LIN {X 0,Y 566.944,Z 607.654,A -85,B 0,C 180,E1 -2597.403,E2 -2597.403} C_VEL
LIN {X 0,Y 566.869,Z 619.609,A -85,B 0,C 180,E1 -2597.674,E2 -2597.674} C_VEL
LIN {X 0,Y 566.746,Z 633.413,A -85,B 0,C 180,E1 -2598.148,E2 -2598.148} C_VEL
LIN {X 0,Y 566.629,Z 645.045,A -85,B 0,C 180,E1 -2598.706,E2 -2598.706} C_VEL
LIN {X 0,Y 566.485,Z 655.838,A -85,B 0,C 180,E1 -2599.366,E2 -2599.366} C_VEL
LIN {X 0,Y 566.315,Z 665.418,A -85,B 0,C 180,E1 -2600.085,E2 -2600.085} C_VEL
LIN {X 0,Y 566.229,Z 674.312,A -85,B 0,C 180,E1 -2600.895,E2 -2600.895} C_VEL
LIN {X 0,Y 566.113,Z 683.962,A -85,B 0,C 180,E1 -2601.972,E2 -2601.972} C_VEL
LIN {X 0,Y 566.009,Z 691.72,A -85,B 0,C 180,E1 -2603.065,E2 -2603.065} C_VEL
LIN {X 0,Y 565.989,Z 696.846,A -85,B 0,C 180,E1 -2603.941,E2 -2603.941} C_VEL
LIN {X 0,Y 565.877,Z 701.915,A -85,B 0,C 180,E1 -2605.013,E2 -2605.013} C_VEL
LIN {X 0,Y 565.927,Z 705.855,A -85,B 0,C 180,E1 -2606.084,E2 -2606.084} C_VEL
LIN {X 0,Y 565.878,Z 708.77,A -85,B 0,C 180,E1 -2607.152,E2 -2607.152} C_VEL
LIN {X 0,Y 565.84,Z 710.209,A -85,B 0,C 180,E1 -2607.865,E2 -2607.865} C_VEL
LIN {X 0,Y 565.841,Z 711.767,A -85,B 0,C 180,E1 -2609.288,E2 -2609.288} C_VEL
LIN {X 0,Y 565.839,Z 712,A -85,B 0,C 180,E1 -2610,E2 -2610} C_VEL
LIN {X 0,Y 565.846,Z 711.177,A -85,B 0,C 180,E1 -2611.423,E2 -2611.423} C_VEL
LIN {X 0,Y 565.84,Z 710.209,A -85,B 0,C 180,E1 -2612.135,E2 -2612.135} C_VEL
LIN {X 0,Y 565.927,Z 706.934,A -85,B 0,C 180,E1 -2613.56,E2 -2613.56} C_VEL
LIN {X 0,Y 565.933,Z 703.334,A -85,B 0,C 180,E1 -2614.63,E2 -2614.63} C_VEL
LIN {X 0,Y 565.998,Z 698.641,A -85,B 0,C 180,E1 -2615.701,E2 -2615.701} C_VEL
LIN {X 0,Y 565.998,Z 692.926,A -85,B 0,C 180,E1 -2616.739,E2 -2616.739} C_VEL
LIN {X 0,Y 566.081,Z 686.651,A -85,B 0,C 180,E1 -2617.67,E2 -2617.67} C_VEL
LIN {X 0,Y 566.174,Z 679.383,A -85,B 0,C 180,E1 -2618.566,E2 -2618.566} C_VEL
LIN {X 0,Y 566.28,Z 670.607,A -85,B 0,C 180,E1 -2619.465,E2 -2619.465} C_VEL
LIN {X 0,Y 566.439,Z 659.729,A -85,B 0,C 180,E1 -2620.364,E2 -2620.364} C_VEL
LIN {X 0,Y 566.591,Z 649.221,A -85,B 0,C 180,E1 -2621.056,E2 -2621.056} C_VEL
LIN {X 0,Y 566.69,Z 638.78,A -85,B 0,C 180,E1 -2621.608,E2 -2621.608} C_VEL
LIN {X 0,Y 566.763,Z 628.631,A -85,B 0,C 180,E1 -2622.033,E2 -2622.033} C_VEL
LIN {X 0,Y 566.923,Z 617.028,A -85,B 0,C 180,E1 -2622.393,E2 -2622.393} C_VEL
LIN {X 0,Y 566.934,Z 605.012,A -85,B 0,C 180,E1 -2622.643,E2 -2622.643} C_VEL
LIN {X 0,Y 567.085,Z 506.315,A -85,B 0,C 180,E1 -2623.906,E2 -2623.906} C_VEL
LIN {X 0,Y 566.329,Z 501.567,A -85,B 0,C 180,E1 -2624.004,E2 -2624.004} C_VEL
LIN {X 0,Y 566.263,Z 499.133,A -85,B 0,C 180,E1 -2624.372,E2 -2624.372} C_VEL
LIN {X 0,Y 566.412,Z 482.577,A -85,B 0,C 180,E1 -2627.325,E2 -2627.325} C_VEL
LIN {X 0,Y 566.641,Z 467.055,A -85,B 0,C 180,E1 -2630.132,E2 -2630.132} C_VEL
LIN {X 0,Y 566.814,Z 451.485,A -85,B 0,C 180,E1 -2632.99,E2 -2632.99} C_VEL
LIN {X 0,Y 566.824,Z 444.171,A -85,B 0,C 180,E1 -2634.347,E2 -2634.347} C_VEL
LIN {X 0,Y 566.177,Z 440.526,A -85,B 0,C 180,E1 -2635.096,E2 -2635.096} C_VEL
LIN {X 0,Y 566.151,Z 440.46,A -85,B 0,C 180,E1 -2637.342,E2 -2637.342} C_VEL
LIN {X 0,Y 566.156,Z 440.462,A -85,B 0,C 180,E1 -2639.771,E2 -2639.771} C_VEL
LIN {X 0,Y 566.178,Z 440.458,A -85,B 0,C 180,E1 -2642.425,E2 -2642.425} C_VEL
LIN {X 0,Y 566.159,Z 440.456,A -85,B 0,C 180,E1 -2644.985,E2 -2644.985} C_VEL
LIN {X 0,Y 566.18,Z 440.454,A -85,B 0,C 180,E1 -2647.462,E2 -2647.462} C_VEL
LIN {X 0,Y 566.159,Z 440.461,A -85,B 0,C 180,E1 -2650.203,E2 -2650.203} C_VEL
LIN {X 0,Y 566.145,Z 440.458,A -85,B 0,C 180,E1 -2653.059,E2 -2653.059} C_VEL
LIN {X 0,Y 566.144,Z 440.466,A -85,B 0,C 180,E1 -2656.054,E2 -2656.054} C_VEL
LIN {X 0,Y 566.133,Z 440.459,A -85,B 0,C 180,E1 -2658.856,E2 -2658.856} C_VEL
LIN {X 0,Y 566.159,Z 440.458,A -85,B 0,C 180,E1 -2661.634,E2 -2661.634} C_VEL
LIN {X 0,Y 566.134,Z 440.464,A -85,B 0,C 180,E1 -2664.305,E2 -2664.305} C_VEL
LIN {X 0,Y 566.16,Z 440.455,A -85,B 0,C 180,E1 -2666.893,E2 -2666.893} C_VEL
LIN {X 0,Y 566.162,Z 440.457,A -85,B 0,C 180,E1 -2669.405,E2 -2669.405} C_VEL
LIN {X 0,Y 566.136,Z 440.464,A -85,B 0,C 180,E1 -2671.852,E2 -2671.852} C_VEL
LIN {X 0,Y 566.172,Z 440.46,A -85,B 0,C 180,E1 -2674.248,E2 -2674.248} C_VEL
LIN {X 0,Y 566.163,Z 440.457,A -85,B 0,C 180,E1 -2676.719,E2 -2676.719} C_VEL
LIN {X 0,Y 566.179,Z 440.453,A -85,B 0,C 180,E1 -2678.9,E2 -2678.9} C_VEL
LIN {X 0,Y 566.151,Z 440.46,A -85,B 0,C 180,E1 -2681.919,E2 -2681.919} C_VEL
LIN {X 0,Y 566.146,Z 440.457,A -85,B 0,C 180,E1 -2684.888,E2 -2684.888} C_VEL
LIN {X 0,Y 566.171,Z 440.46,A -85,B 0,C 180,E1 -2687.817,E2 -2687.817} C_VEL
LIN {X 0,Y 566.149,Z 440.463,A -85,B 0,C 180,E1 -2689.991,E2 -2689.991} C_VEL
LIN {X 0,Y 566.177,Z 440.453,A -85,B 0,C 180,E1 -2692.868,E2 -2692.868} C_VEL
LIN {X 0,Y 566.242,Z 440.446,A -85,B 0,C 180,E1 -2695.015,E2 -2695.015} C_VEL
LIN {X 0,Y 566.273,Z 440.448,A -85,B 0,C 180,E1 -2697.865,E2 -2697.865} C_VEL
LIN {X 0,Y 566.279,Z 440.446,A -85,B 0,C 180,E1 -2699.999,E2 -2699.999} C_VEL
LIN {X 0,Y 566.231,Z 440.446,A -85,B 0,C 180,E1 -2702.845,E2 -2702.845} C_VEL
LIN {X 0,Y 566.226,Z 440.452,A -85,B 0,C 180,E1 -2705.697,E2 -2705.697} C_VEL
LIN {X 0,Y 566.178,Z 440.453,A -85,B 0,C 180,E1 -2708.565,E2 -2708.565} C_VEL
LIN {X 0,Y 566.185,Z 440.451,A -85,B 0,C 180,E1 -2711.454,E2 -2711.454} C_VEL
LIN {X 0,Y 566.2,Z 440.454,A -85,B 0,C 180,E1 -2714.495,E2 -2714.495} C_VEL
LIN {X 0,Y 566.142,Z 440.458,A -85,B 0,C 180,E1 -2717.332,E2 -2717.332} C_VEL
LIN {X 0,Y 566.158,Z 440.46,A -85,B 0,C 180,E1 -2720.338,E2 -2720.338} C_VEL
LIN {X 0,Y 566.148,Z 440.459,A -85,B 0,C 180,E1 -2722.631,E2 -2722.631} C_VEL
LIN {X 0,Y 566.167,Z 440.454,A -85,B 0,C 180,E1 -2725.02,E2 -2725.02} C_VEL
LIN {X 0,Y 566.139,Z 440.456,A -85,B 0,C 180,E1 -2727.445,E2 -2727.445} C_VEL
LIN {X 0,Y 565.453,Z 440.55,A -85,B 0,C 180,E1 -2728.039,E2 -2728.039} C_VEL
LIN {X 0,Y 562.598,Z 440.907,A -85,B 0,C 180,E1 -2729.003,E2 -2729.003} C_VEL
LIN {X 0,Y 560.205,Z 441.205,A -85,B 0,C 180,E1 -2729.779,E2 -2729.779} C_VEL
LIN {X 0,Y 559.188,Z 441.33,A -85,B 0,C 180,E1 -2730.378,E2 -2730.378} C_VEL
LIN {X 0,Y 559.111,Z 441.337,A -85,B 0,C 180,E1 -2730.581,E2 -2730.581} C_VEL
LIN {X 0,Y 559.122,Z 441.333,A -85,B 0,C 180,E1 -2732.716,E2 -2732.716} C_VEL
LIN {X 0,Y 559.1,Z 441.333,A -85,B 0,C 180,E1 -2735.324,E2 -2735.324} C_VEL
LIN {X 0,Y 559.108,Z 441.344,A -85,B 0,C 180,E1 -2738.018,E2 -2738.018} C_VEL
LIN {X 0,Y 559.111,Z 441.332,A -85,B 0,C 180,E1 -2740.814,E2 -2740.814} C_VEL
LIN {X 0,Y 559.085,Z 441.338,A -85,B 0,C 180,E1 -2743.19,E2 -2743.19} C_VEL
LIN {X 0,Y 559.107,Z 441.339,A -85,B 0,C 180,E1 -2745.763,E2 -2745.763} C_VEL
LIN {X 0,Y 559.082,Z 441.339,A -85,B 0,C 180,E1 -2748.223,E2 -2748.223} C_VEL
LIN {X 0,Y 559.152,Z 441.329,A -85,B 0,C 180,E1 -2751.192,E2 -2751.192} C_VEL
LIN {X 0,Y 559.095,Z 441.342,A -85,B 0,C 180,E1 -2753.786,E2 -2753.786} C_VEL
LIN {X 0,Y 559.119,Z 441.336,A -85,B 0,C 180,E1 -2756.423,E2 -2756.423} C_VEL
LIN {X 0,Y 559.13,Z 441.332,A -85,B 0,C 180,E1 -2758.98,E2 -2758.98} C_VEL
LIN {X 0,Y 559.09,Z 441.338,A -85,B 0,C 180,E1 -2761.63,E2 -2761.63} C_VEL
LIN {X 0,Y 559.131,Z 441.34,A -85,B 0,C 180,E1 -2763.901,E2 -2763.901} C_VEL
LIN {X 0,Y 559.093,Z 441.337,A -85,B 0,C 180,E1 -2767.066,E2 -2767.066} C_VEL
LIN {X 0,Y 559.144,Z 441.332,A -85,B 0,C 180,E1 -2769.394,E2 -2769.394} C_VEL
LIN {X 0,Y 559.099,Z 441.341,A -85,B 0,C 180,E1 -2771.684,E2 -2771.684} C_VEL
LIN {X 0,Y 559.113,Z 441.336,A -85,B 0,C 180,E1 -2774.695,E2 -2774.695} C_VEL
LIN {X 0,Y 559.123,Z 441.334,A -85,B 0,C 180,E1 -2776.924,E2 -2776.924} C_VEL
LIN {X 0,Y 559.15,Z 441.331,A -85,B 0,C 180,E1 -2779.133,E2 -2779.133} C_VEL
LIN {X 0,Y 559.124,Z 441.342,A -85,B 0,C 180,E1 -2782.053,E2 -2782.053} C_VEL
LIN {X 0,Y 559.21,Z 441.323,A -85,B 0,C 180,E1 -2784.953,E2 -2784.953} C_VEL
LIN {X 0,Y 559.235,Z 441.327,A -85,B 0,C 180,E1 -2787.839,E2 -2787.839} C_VEL
LIN {X 0,Y 559.238,Z 441.328,A -85,B 0,C 180,E1 -2790,E2 -2790} C_VEL
LIN {X 0,Y 559.19,Z 441.326,A -85,B 0,C 180,E1 -2792.882,E2 -2792.882} C_VEL
LIN {X 0,Y 559.19,Z 441.332,A -85,B 0,C 180,E1 -2795.771,E2 -2795.771} C_VEL
LIN {X 0,Y 559.141,Z 441.333,A -85,B 0,C 180,E1 -2798.675,E2 -2798.675} C_VEL
LIN {X 0,Y 559.138,Z 441.336,A -85,B 0,C 180,E1 -2801.602,E2 -2801.602} C_VEL
LIN {X 0,Y 559.164,Z 441.33,A -85,B 0,C 180,E1 -2804.588,E2 -2804.588} C_VEL
LIN {X 0,Y 559.096,Z 441.34,A -85,B 0,C 180,E1 -2807.559,E2 -2807.559} C_VEL
LIN {X 0,Y 559.142,Z 441.339,A -85,B 0,C 180,E1 -2809.838,E2 -2809.838} C_VEL
LIN {X 0,Y 559.111,Z 441.342,A -85,B 0,C 180,E1 -2812.154,E2 -2812.154} C_VEL
LIN {X 0,Y 559.121,Z 441.334,A -85,B 0,C 180,E1 -2815.178,E2 -2815.178} C_VEL
LIN {X 0,Y 559.087,Z 441.343,A -85,B 0,C 180,E1 -2817.717,E2 -2817.717} C_VEL
LIN {X 0,Y 559.114,Z 441.34,A -85,B 0,C 180,E1 -2820.185,E2 -2820.185} C_VEL
LIN {X 0,Y 559.118,Z 441.333,A -85,B 0,C 180,E1 -2822.717,E2 -2822.717} C_VEL
LIN {X 0,Y 559.097,Z 441.332,A -85,B 0,C 180,E1 -2825.326,E2 -2825.326} C_VEL
LIN {X 0,Y 559.106,Z 441.344,A -85,B 0,C 180,E1 -2828.019,E2 -2828.019} C_VEL
LIN {X 0,Y 559.108,Z 441.341,A -85,B 0,C 180,E1 -2829.938,E2 -2829.938} C_VEL
LIN {X 0,Y 559.098,Z 441.33,A -85,B 0,C 180,E1 -2832.749,E2 -2832.749} C_VEL
LIN {X 0,Y 559.108,Z 441.34,A -85,B 0,C 180,E1 -2835.765,E2 -2835.765} C_VEL
LIN {X 0,Y 559.103,Z 441.338,A -85,B 0,C 180,E1 -2838.226,E2 -2838.226} C_VEL
LIN {X 0,Y 559.154,Z 441.329,A -85,B 0,C 180,E1 -2841.194,E2 -2841.194} C_VEL
LIN {X 0,Y 559.098,Z 441.343,A -85,B 0,C 180,E1 -2843.788,E2 -2843.788} C_VEL
LIN {X 0,Y 559.123,Z 441.335,A -85,B 0,C 180,E1 -2846.424,E2 -2846.424} C_VEL
LIN {X 0,Y 559.134,Z 441.331,A -85,B 0,C 180,E1 -2848.981,E2 -2848.981} C_VEL
LIN {X 0,Y 559.095,Z 441.339,A -85,B 0,C 180,E1 -2851.632,E2 -2851.632} C_VEL
LIN {X 0,Y 559.11,Z 441.334,A -85,B 0,C 180,E1 -2854.7,E2 -2854.7} C_VEL
LIN {X 0,Y 559.099,Z 441.336,A -85,B 0,C 180,E1 -2857.067,E2 -2857.067} C_VEL
LIN {X 0,Y 559.137,Z 441.331,A -85,B 0,C 180,E1 -2859.395,E2 -2859.395} C_VEL
LIN {X 0,Y 559.097,Z 441.337,A -85,B 0,C 180,E1 -2862.442,E2 -2862.442} C_VEL
LIN {X 0,Y 559.149,Z 441.332,A -85,B 0,C 180,E1 -2865.442,E2 -2865.442} C_VEL
LIN {X 0,Y 559.147,Z 441.328,A -85,B 0,C 180,E1 -2868.4,E2 -2868.4} C_VEL
LIN {X 0,Y 559.142,Z 441.328,A -85,B 0,C 180,E1 -2871.326,E2 -2871.326} C_VEL
LIN {X 0,Y 559.196,Z 441.329,A -85,B 0,C 180,E1 -2874.231,E2 -2874.231} C_VEL
LIN {X 0,Y 559.241,Z 441.325,A -85,B 0,C 180,E1 -2877.841,E2 -2877.841} C_VEL
LIN {X 0,Y 559.247,Z 441.321,A -85,B 0,C 180,E1 -2880.001,E2 -2880.001} C_VEL
LIN {X 0,Y 559.198,Z 441.322,A -85,B 0,C 180,E1 -2882.883,E2 -2882.883} C_VEL
LIN {X 0,Y 559.197,Z 441.331,A -85,B 0,C 180,E1 -2885.772,E2 -2885.772} C_VEL
LIN {X 0,Y 559.145,Z 441.325,A -85,B 0,C 180,E1 -2888.676,E2 -2888.676} C_VEL
LIN {X 0,Y 559.151,Z 441.331,A -85,B 0,C 180,E1 -2891.603,E2 -2891.603} C_VEL
LIN {X 0,Y 559.149,Z 441.33,A -85,B 0,C 180,E1 -2894.577,E2 -2894.577} C_VEL
LIN {X 0,Y 559.103,Z 441.336,A -85,B 0,C 180,E1 -2897.56,E2 -2897.56} C_VEL
LIN {X 0,Y 559.104,Z 441.334,A -85,B 0,C 180,E1 -2900.608,E2 -2900.608} C_VEL
LIN {X 0,Y 559.129,Z 441.334,A -85,B 0,C 180,E1 -2903.427,E2 -2903.427} C_VEL
LIN {X 0,Y 559.14,Z 441.333,A -85,B 0,C 180,E1 -2906.1,E2 -2906.1} C_VEL
LIN {X 0,Y 559.096,Z 441.337,A -85,B 0,C 180,E1 -2908.534,E2 -2908.534} C_VEL
LIN {X 0,Y 559.135,Z 441.332,A -85,B 0,C 180,E1 -2911.272,E2 -2911.272} C_VEL
LIN {X 0,Y 559.149,Z 441.335,A -85,B 0,C 180,E1 -2913.947,E2 -2913.947} C_VEL
LIN {X 0,Y 559.108,Z 441.335,A -85,B 0,C 180,E1 -2917.112,E2 -2917.112} C_VEL
LIN {X 0,Y 559.119,Z 441.341,A -85,B 0,C 180,E1 -2919.937,E2 -2919.937} C_VEL
LIN {X 0,Y 559.108,Z 441.335,A -85,B 0,C 180,E1 -2922.749,E2 -2922.749} C_VEL
LIN {X 0,Y 559.12,Z 441.341,A -85,B 0,C 180,E1 -2925.765,E2 -2925.765} C_VEL
LIN {X 0,Y 559.095,Z 441.337,A -85,B 0,C 180,E1 -2928.224,E2 -2928.224} C_VEL
LIN {X 0,Y 559.167,Z 441.328,A -85,B 0,C 180,E1 -2931.194,E2 -2931.194} C_VEL
LIN {X 0,Y 559.106,Z 441.341,A -85,B 0,C 180,E1 -2933.787,E2 -2933.787} C_VEL
LIN {X 0,Y 559.124,Z 441.334,A -85,B 0,C 180,E1 -2936.423,E2 -2936.423} C_VEL
LIN {X 0,Y 559.14,Z 441.332,A -85,B 0,C 180,E1 -2938.98,E2 -2938.98} C_VEL
LIN {X 0,Y 559.101,Z 441.343,A -85,B 0,C 180,E1 -2941.633,E2 -2941.633} C_VEL
LIN {X 0,Y 559.149,Z 441.399,A -85,B 0,C 180,E1 -2944.751,E2 -2944.751} C_VEL
LIN {X 0,Y 559.952,Z 447.174,A -85,B 0,C 180,E1 -2945.927,E2 -2945.927} C_VEL
LIN {X 0,Y 559.722,Z 463.918,A -85,B 0,C 180,E1 -2949.032,E2 -2949.032} C_VEL
LIN {X 0,Y 559.496,Z 481.542,A -85,B 0,C 180,E1 -2952.265,E2 -2952.265} C_VEL
LIN {X 0,Y 559.24,Z 499.133,A -85,B 0,C 180,E1 -2955.443,E2 -2955.443} C_VEL
LIN {X 0,Y 559.283,Z 501.579,A -85,B 0,C 180,E1 -2955.816,E2 -2955.816} C_VEL
LIN {X 0,Y 560.229,Z 507.309,A -85,B 0,C 180,E1 -2955.933,E2 -2955.933} C_VEL
LIN {X 0,Y 560.033,Z 607.603,A -85,B 0,C 180,E1 -2957.245,E2 -2957.245} C_VEL
LIN {X 0,Y 559.963,Z 618.717,A -85,B 0,C 180,E1 -2957.496,E2 -2957.496} C_VEL
LIN {X 0,Y 559.817,Z 631.133,A -85,B 0,C 180,E1 -2957.908,E2 -2957.908} C_VEL
LIN {X 0,Y 559.67,Z 644.741,A -85,B 0,C 180,E1 -2958.547,E2 -2958.547} C_VEL
LIN {X 0,Y 559.537,Z 654.514,A -85,B 0,C 180,E1 -2959.14,E2 -2959.14} C_VEL
LIN {X 0,Y 559.356,Z 664.311,A -85,B 0,C 180,E1 -2959.869,E2 -2959.869} C_VEL
LIN {X 0,Y 559.237,Z 672.456,A -85,B 0,C 180,E1 -2960.597,E2 -2960.597} C_VEL
LIN {X 0,Y 559.113,Z 680.928,A -85,B 0,C 180,E1 -2961.507,E2 -2961.507} C_VEL
LIN {X 0,Y 558.996,Z 687.948,A -85,B 0,C 180,E1 -2962.414,E2 -2962.414} C_VEL
LIN {X 0,Y 558.894,Z 694.873,A -85,B 0,C 180,E1 -2963.502,E2 -2963.502} C_VEL
LIN {X 0,Y 558.868,Z 700.383,A -85,B 0,C 180,E1 -2964.588,E2 -2964.588} C_VEL
LIN {X 0,Y 558.869,Z 704.694,A -85,B 0,C 180,E1 -2965.673,E2 -2965.673} C_VEL
LIN {X 0,Y 558.799,Z 708.763,A -85,B 0,C 180,E1 -2967.116,E2 -2967.116} C_VEL
LIN {X 0,Y 558.746,Z 710.21,A -85,B 0,C 180,E1 -2967.837,E2 -2967.837} C_VEL
LIN {X 0,Y 558.741,Z 711.759,A -85,B 0,C 180,E1 -2969.279,E2 -2969.279} C_VEL
LIN {X 0,Y 558.74,Z 712,A -85,B 0,C 180,E1 -2970,E2 -2970} C_VEL
LIN {X 0,Y 558.745,Z 711.169,A -85,B 0,C 180,E1 -2971.441,E2 -2971.441} C_VEL
LIN {X 0,Y 558.746,Z 710.21,A -85,B 0,C 180,E1 -2972.163,E2 -2972.163} C_VEL
LIN {X 0,Y 558.836,Z 706.929,A -85,B 0,C 180,E1 -2973.605,E2 -2973.605} C_VEL
LIN {X 0,Y 558.826,Z 703.328,A -85,B 0,C 180,E1 -2974.689,E2 -2974.689} C_VEL
LIN {X 0,Y 558.929,Z 698.633,A -85,B 0,C 180,E1 -2975.773,E2 -2975.773} C_VEL
LIN {X 0,Y 558.925,Z 692.918,A -85,B 0,C 180,E1 -2976.824,E2 -2976.824} C_VEL
LIN {X 0,Y 559.009,Z 686.642,A -85,B 0,C 180,E1 -2977.767,E2 -2977.767} C_VEL
LIN {X 0,Y 559.105,Z 679.373,A -85,B 0,C 180,E1 -2978.676,E2 -2978.676} C_VEL
LIN {X 0,Y 559.241,Z 670.607,A -85,B 0,C 180,E1 -2979.585,E2 -2979.585} C_VEL
LIN {X 0,Y 559.427,Z 659.726,A -85,B 0,C 180,E1 -2980.496,E2 -2980.496} C_VEL
LIN {X 0,Y 559.609,Z 649.543,A -85,B 0,C 180,E1 -2981.176,E2 -2981.176} C_VEL
LIN {X 0,Y 559.729,Z 638.765,A -85,B 0,C 180,E1 -2981.754,E2 -2981.754} C_VEL
LIN {X 0,Y 559.833,Z 628.609,A -85,B 0,C 180,E1 -2982.184,E2 -2982.184} C_VEL
LIN {X 0,Y 559.985,Z 617.857,A -85,B 0,C 180,E1 -2982.526,E2 -2982.526} C_VEL
LIN {X 0,Y 560.033,Z 607.603,A -85,B 0,C 180,E1 -2982.755,E2 -2982.755} C_VEL
LIN {X 0,Y 560.224,Z 507.309,A -85,B 0,C 180,E1 -2984.067,E2 -2984.067} C_VEL
LIN {X 0,Y 559.283,Z 501.577,A -85,B 0,C 180,E1 -2984.184,E2 -2984.184} C_VEL
LIN {X 0,Y 559.24,Z 499.133,A -85,B 0,C 180,E1 -2984.557,E2 -2984.557} C_VEL
LIN {X 0,Y 559.496,Z 481.542,A -85,B 0,C 180,E1 -2987.735,E2 -2987.735} C_VEL
LIN {X 0,Y 559.722,Z 463.918,A -85,B 0,C 180,E1 -2990.968,E2 -2990.968} C_VEL
LIN {X 0,Y 559.963,Z 447.2,A -85,B 0,C 180,E1 -2994.073,E2 -2994.073} C_VEL
LIN {X 0,Y 559.149,Z 441.399,A -85,B 0,C 180,E1 -2995.249,E2 -2995.249} C_VEL
LIN {X 0,Y 559.101,Z 441.343,A -85,B 0,C 180,E1 -2998.367,E2 -2998.367} C_VEL
LIN {X 0,Y 559.122,Z 441.334,A -85,B 0,C 180,E1 -3001.268,E2 -3001.268} C_VEL
LIN {X 0,Y 559.151,Z 441.336,A -85,B 0,C 180,E1 -3003.946,E2 -3003.946} C_VEL
LIN {X 0,Y 559.105,Z 441.334,A -85,B 0,C 180,E1 -3007.111,E2 -3007.111} C_VEL
LIN {X 0,Y 559.144,Z 441.336,A -85,B 0,C 180,E1 -3009.868,E2 -3009.868} C_VEL
LIN {X 0,Y 559.112,Z 441.335,A -85,B 0,C 180,E1 -3012.748,E2 -3012.748} C_VEL
LIN {X 0,Y 559.119,Z 441.333,A -85,B 0,C 180,E1 -3015.258,E2 -3015.258} C_VEL
LIN {X 0,Y 559.093,Z 441.344,A -85,B 0,C 180,E1 -3018.223,E2 -3018.223} C_VEL
LIN {X 0,Y 559.135,Z 441.33,A -85,B 0,C 180,E1 -3021.196,E2 -3021.196} C_VEL
LIN {X 0,Y 559.109,Z 441.339,A -85,B 0,C 180,E1 -3023.786,E2 -3023.786} C_VEL
LIN {X 0,Y 559.134,Z 441.334,A -85,B 0,C 180,E1 -3026.422,E2 -3026.422} C_VEL
LIN {X 0,Y 559.144,Z 441.33,A -85,B 0,C 180,E1 -3028.979,E2 -3028.979} C_VEL
LIN {X 0,Y 559.099,Z 441.338,A -85,B 0,C 180,E1 -3031.631,E2 -3031.631} C_VEL
LIN {X 0,Y 559.119,Z 441.333,A -85,B 0,C 180,E1 -3034.698,E2 -3034.698} C_VEL
LIN {X 0,Y 559.107,Z 441.334,A -85,B 0,C 180,E1 -3037.065,E2 -3037.065} C_VEL
LIN {X 0,Y 559.104,Z 441.334,A -85,B 0,C 180,E1 -3039.392,E2 -3039.392} C_VEL
LIN {X 0,Y 559.103,Z 441.336,A -85,B 0,C 180,E1 -3042.44,E2 -3042.44} C_VEL
LIN {X 0,Y 559.147,Z 441.33,A -85,B 0,C 180,E1 -3045.44,E2 -3045.44} C_VEL
LIN {X 0,Y 559.151,Z 441.331,A -85,B 0,C 180,E1 -3048.397,E2 -3048.397} C_VEL
LIN {X 0,Y 559.145,Z 441.325,A -85,B 0,C 180,E1 -3051.324,E2 -3051.324} C_VEL
LIN {X 0,Y 559.197,Z 441.331,A -85,B 0,C 180,E1 -3054.228,E2 -3054.228} C_VEL
LIN {X 0,Y 559.243,Z 441.323,A -85,B 0,C 180,E1 -3057.838,E2 -3057.838} C_VEL
LIN {X 0,Y 559.248,Z 441.321,A -85,B 0,C 180,E1 -3059.999,E2 -3059.999} C_VEL
LIN {X 0,Y 559.198,Z 441.322,A -85,B 0,C 180,E1 -3062.88,E2 -3062.88} C_VEL
LIN {X 0,Y 559.196,Z 441.329,A -85,B 0,C 180,E1 -3065.769,E2 -3065.769} C_VEL
LIN {X 0,Y 559.142,Z 441.328,A -85,B 0,C 180,E1 -3068.674,E2 -3068.674} C_VEL
LIN {X 0,Y 559.147,Z 441.328,A -85,B 0,C 180,E1 -3071.6,E2 -3071.6} C_VEL
LIN {X 0,Y 559.147,Z 441.332,A -85,B 0,C 180,E1 -3074.576,E2 -3074.576} C_VEL
LIN {X 0,Y 559.098,Z 441.337,A -85,B 0,C 180,E1 -3077.557,E2 -3077.557} C_VEL
LIN {X 0,Y 559.137,Z 441.331,A -85,B 0,C 180,E1 -3080.605,E2 -3080.605} C_VEL
LIN {X 0,Y 559.122,Z 441.334,A -85,B 0,C 180,E1 -3083.425,E2 -3083.425} C_VEL
LIN {X 0,Y 559.13,Z 441.337,A -85,B 0,C 180,E1 -3086.098,E2 -3086.098} C_VEL
LIN {X 0,Y 559.091,Z 441.338,A -85,B 0,C 180,E1 -3088.532,E2 -3088.532} C_VEL
LIN {X 0,Y 559.111,Z 441.337,A -85,B 0,C 180,E1 -3090.581,E2 -3090.581} C_VEL
LIN {X 0,Y 558.454,Z 441.418,A -85,B 0,C 180,E1 -3091.182,E2 -3091.182} C_VEL
LIN {X 0,Y 555.592,Z 441.78,A -85,B 0,C 180,E1 -3092.158,E2 -3092.158} C_VEL
LIN {X 0,Y 553.173,Z 442.076,A -85,B 0,C 180,E1 -3092.944,E2 -3092.944} C_VEL
LIN {X 0,Y 552.145,Z 442.203,A -85,B 0,C 180,E1 -3093.55,E2 -3093.55} C_VEL
LIN {X 0,Y 552.067,Z 442.213,A -85,B 0,C 180,E1 -3093.756,E2 -3093.756} C_VEL
LIN {X 0,Y 552.037,Z 442.216,A -85,B 0,C 180,E1 -3096.75,E2 -3096.75} C_VEL
LIN {X 0,Y 552.111,Z 442.208,A -85,B 0,C 180,E1 -3099.527,E2 -3099.527} C_VEL
LIN {X 0,Y 552.068,Z 442.215,A -85,B 0,C 180,E1 -3102.429,E2 -3102.429} C_VEL
LIN {X 0,Y 552.058,Z 442.214,A -85,B 0,C 180,E1 -3105.559,E2 -3105.559} C_VEL
LIN {X 0,Y 552.037,Z 442.212,A -85,B 0,C 180,E1 -3108.547,E2 -3108.547} C_VEL
LIN {X 0,Y 552.094,Z 442.21,A -85,B 0,C 180,E1 -3111.41,E2 -3111.41} C_VEL
LIN {X 0,Y 552.045,Z 442.211,A -85,B 0,C 180,E1 -3114.562,E2 -3114.562} C_VEL
LIN {X 0,Y 552.08,Z 442.21,A -85,B 0,C 180,E1 -3117.156,E2 -3117.156} C_VEL
LIN {X 0,Y 552.072,Z 442.217,A -85,B 0,C 180,E1 -3119.954,E2 -3119.954} C_VEL
LIN {X 0,Y 552.06,Z 442.213,A -85,B 0,C 180,E1 -3123.012,E2 -3123.012} C_VEL
LIN {X 0,Y 552.058,Z 442.222,A -85,B 0,C 180,E1 -3125.96,E2 -3125.96} C_VEL
LIN {X 0,Y 552.073,Z 442.217,A -85,B 0,C 180,E1 -3128.335,E2 -3128.335} C_VEL
LIN {X 0,Y 552.12,Z 442.207,A -85,B 0,C 180,E1 -3130.673,E2 -3130.673} C_VEL
LIN {X 0,Y 552.055,Z 442.22,A -85,B 0,C 180,E1 -3133.736,E2 -3133.736} C_VEL
LIN {X 0,Y 552.103,Z 442.217,A -85,B 0,C 180,E1 -3136.004,E2 -3136.004} C_VEL
LIN {X 0,Y 552.11,Z 442.208,A -85,B 0,C 180,E1 -3138.992,E2 -3138.992} C_VEL
LIN {X 0,Y 552.093,Z 442.218,A -85,B 0,C 180,E1 -3141.951,E2 -3141.951} C_VEL
LIN {X 0,Y 552.187,Z 442.198,A -85,B 0,C 180,E1 -3144.889,E2 -3144.889} C_VEL
LIN {X 0,Y 552.205,Z 442.203,A -85,B 0,C 180,E1 -3147.812,E2 -3147.812} C_VEL
LIN {X 0,Y 552.207,Z 442.204,A -85,B 0,C 180,E1 -3150,E2 -3150} C_VEL
LIN {X 0,Y 552.158,Z 442.202,A -85,B 0,C 180,E1 -3152.918,E2 -3152.918} C_VEL
LIN {X 0,Y 552.161,Z 442.209,A -85,B 0,C 180,E1 -3155.844,E2 -3155.844} C_VEL
LIN {X 0,Y 552.113,Z 442.208,A -85,B 0,C 180,E1 -3158.786,E2 -3158.786} C_VEL
LIN {X 0,Y 552.084,Z 442.217,A -85,B 0,C 180,E1 -3161.752,E2 -3161.752} C_VEL
LIN {X 0,Y 552.111,Z 442.208,A -85,B 0,C 180,E1 -3164.749,E2 -3164.749} C_VEL
LIN {X 0,Y 552.06,Z 442.22,A -85,B 0,C 180,E1 -3167.79,E2 -3167.79} C_VEL
LIN {X 0,Y 552.101,Z 442.216,A -85,B 0,C 180,E1 -3170.102,E2 -3170.102} C_VEL
LIN {X 0,Y 552.064,Z 442.216,A -85,B 0,C 180,E1 -3172.452,E2 -3172.452} C_VEL
LIN {X 0,Y 552.063,Z 442.214,A -85,B 0,C 180,E1 -3175.334,E2 -3175.334} C_VEL
LIN {X 0,Y 552.036,Z 442.221,A -85,B 0,C 180,E1 -3178.102,E2 -3178.102} C_VEL
LIN {X 0,Y 552.073,Z 442.212,A -85,B 0,C 180,E1 -3180.611,E2 -3180.611} C_VEL
LIN {X 0,Y 552.078,Z 442.21,A -85,B 0,C 180,E1 -3183.188,E2 -3183.188} C_VEL
LIN {X 0,Y 552.05,Z 442.216,A -85,B 0,C 180,E1 -3185.846,E2 -3185.846} C_VEL
LIN {X 0,Y 552.094,Z 442.21,A -85,B 0,C 180,E1 -3188.59,E2 -3188.59} C_VEL
LIN {X 0,Y 552.037,Z 442.212,A -85,B 0,C 180,E1 -3191.453,E2 -3191.453} C_VEL
LIN {X 0,Y 552.059,Z 442.213,A -85,B 0,C 180,E1 -3194.53,E2 -3194.53} C_VEL
LIN {X 0,Y 552.069,Z 442.216,A -85,B 0,C 180,E1 -3197.591,E2 -3197.591} C_VEL
LIN {X 0,Y 552.111,Z 442.208,A -85,B 0,C 180,E1 -3200.473,E2 -3200.473} C_VEL
LIN {X 0,Y 552.036,Z 442.217,A -85,B 0,C 180,E1 -3203.326,E2 -3203.326} C_VEL
LIN {X 0,Y 552.082,Z 442.215,A -85,B 0,C 180,E1 -3205.938,E2 -3205.938} C_VEL
LIN {X 0,Y 552.091,Z 442.211,A -85,B 0,C 180,E1 -3208.541,E2 -3208.541} C_VEL
LIN {X 0,Y 552.062,Z 442.213,A -85,B 0,C 180,E1 -3211.449,E2 -3211.449} C_VEL
LIN {X 0,Y 552.062,Z 442.215,A -85,B 0,C 180,E1 -3214.354,E2 -3214.354} C_VEL
LIN {X 0,Y 552.078,Z 442.211,A -85,B 0,C 180,E1 -3216.758,E2 -3216.758} C_VEL
LIN {X 0,Y 552.085,Z 442.207,A -85,B 0,C 180,E1 -3219.12,E2 -3219.12} C_VEL
LIN {X 0,Y 552.044,Z 442.211,A -85,B 0,C 180,E1 -3221.443,E2 -3221.443} C_VEL
LIN {X 0,Y 552.059,Z 442.217,A -85,B 0,C 180,E1 -3223.737,E2 -3223.737} C_VEL
LIN {X 0,Y 552.099,Z 442.216,A -85,B 0,C 180,E1 -3226.005,E2 -3226.005} C_VEL
LIN {X 0,Y 552.116,Z 442.201,A -85,B 0,C 180,E1 -3228.994,E2 -3228.994} C_VEL
LIN {X 0,Y 552.1,Z 442.214,A -85,B 0,C 180,E1 -3231.952,E2 -3231.952} C_VEL
LIN {X 0,Y 552.194,Z 442.196,A -85,B 0,C 180,E1 -3234.89,E2 -3234.89} C_VEL
LIN {X 0,Y 552.212,Z 442.2,A -85,B 0,C 180,E1 -3237.813,E2 -3237.813} C_VEL
LIN {X 0,Y 552.216,Z 442.196,A -85,B 0,C 180,E1 -3240.001,E2 -3240.001} C_VEL
LIN {X 0,Y 552.166,Z 442.198,A -85,B 0,C 180,E1 -3242.919,E2 -3242.919} C_VEL
LIN {X 0,Y 552.167,Z 442.208,A -85,B 0,C 180,E1 -3245.845,E2 -3245.845} C_VEL
LIN {X 0,Y 552.118,Z 442.199,A -85,B 0,C 180,E1 -3248.787,E2 -3248.787} C_VEL
LIN {X 0,Y 552.097,Z 442.211,A -85,B 0,C 180,E1 -3251.753,E2 -3251.753} C_VEL
LIN {X 0,Y 552.085,Z 442.209,A -85,B 0,C 180,E1 -3254.751,E2 -3254.751} C_VEL
LIN {X 0,Y 552.064,Z 442.216,A -85,B 0,C 180,E1 -3257.791,E2 -3257.791} C_VEL
LIN {X 0,Y 552.045,Z 442.22,A -85,B 0,C 180,E1 -3260.105,E2 -3260.105} C_VEL
LIN {X 0,Y 552.077,Z 442.212,A -85,B 0,C 180,E1 -3262.453,E2 -3262.453} C_VEL
LIN {X 0,Y 552.076,Z 442.21,A -85,B 0,C 180,E1 -3265.334,E2 -3265.334} C_VEL
LIN {X 0,Y 552.044,Z 442.22,A -85,B 0,C 180,E1 -3268.103,E2 -3268.103} C_VEL
LIN {X 0,Y 552.087,Z 442.21,A -85,B 0,C 180,E1 -3270.611,E2 -3270.611} C_VEL
LIN {X 0,Y 552.093,Z 442.207,A -85,B 0,C 180,E1 -3273.188,E2 -3273.188} C_VEL
LIN {X 0,Y 552.064,Z 442.219,A -85,B 0,C 180,E1 -3275.846,E2 -3275.846} C_VEL
LIN {X 0,Y 552.086,Z 442.209,A -85,B 0,C 180,E1 -3278.592,E2 -3278.592} C_VEL
LIN {X 0,Y 552.05,Z 442.216,A -85,B 0,C 180,E1 -3281.453,E2 -3281.453} C_VEL
LIN {X 0,Y 552.067,Z 442.213,A -85,B 0,C 180,E1 -3284.529,E2 -3284.529} C_VEL
LIN {X 0,Y 552.08,Z 442.215,A -85,B 0,C 180,E1 -3287.591,E2 -3287.591} C_VEL
LIN {X 0,Y 552.111,Z 442.206,A -85,B 0,C 180,E1 -3290.941,E2 -3290.941} C_VEL
LIN {X 0,Y 552.047,Z 442.216,A -85,B 0,C 180,E1 -3293.326,E2 -3293.326} C_VEL
LIN {X 0,Y 552.086,Z 442.218,A -85,B 0,C 180,E1 -3295.937,E2 -3295.937} C_VEL
LIN {X 0,Y 552.081,Z 442.213,A -85,B 0,C 180,E1 -3298.539,E2 -3298.539} C_VEL
LIN {X 0,Y 552.07,Z 442.217,A -85,B 0,C 180,E1 -3301.449,E2 -3301.449} C_VEL
LIN {X 0,Y 552.118,Z 442.309,A -85,B 0,C 180,E1 -3304.621,E2 -3304.621} C_VEL
LIN {X 0,Y 553.002,Z 448.119,A -85,B 0,C 180,E1 -3305.804,E2 -3305.804} C_VEL
LIN {X 0,Y 552.719,Z 462.732,A -85,B 0,C 180,E1 -3308.558,E2 -3308.558} C_VEL
LIN {X 0,Y 552.528,Z 476.336,A -85,B 0,C 180,E1 -3311.074,E2 -3311.074} C_VEL
LIN {X 0,Y 552.347,Z 488.785,A -85,B 0,C 180,E1 -3313.364,E2 -3313.364} C_VEL
LIN {X 0,Y 552.217,Z 501.24,A -85,B 0,C 180,E1 -3315.605,E2 -3315.605} C_VEL
LIN {X 0,Y 552.544,Z 503.439,A -85,B 0,C 180,E1 -3315.683,E2 -3315.683} C_VEL
LIN {X 0,Y 553.383,Z 509.309,A -85,B 0,C 180,E1 -3315.782,E2 -3315.782} C_VEL
LIN {X 0,Y 553.098,Z 606.231,A -85,B 0,C 180,E1 -3317.059,E2 -3317.059} C_VEL
LIN {X 0,Y 553.052,Z 616.964,A -85,B 0,C 180,E1 -3317.291,E2 -3317.291} C_VEL
LIN {X 0,Y 552.902,Z 627.575,A -85,B 0,C 180,E1 -3317.623,E2 -3317.623} C_VEL
LIN {X 0,Y 552.78,Z 637.155,A -85,B 0,C 180,E1 -3318.02,E2 -3318.02} C_VEL
LIN {X 0,Y 552.682,Z 646.618,A -85,B 0,C 180,E1 -3318.511,E2 -3318.511} C_VEL
LIN {X 0,Y 552.511,Z 655.811,A -85,B 0,C 180,E1 -3319.093,E2 -3319.093} C_VEL
LIN {X 0,Y 552.361,Z 664.298,A -85,B 0,C 180,E1 -3319.739,E2 -3319.739} C_VEL
LIN {X 0,Y 552.199,Z 672.444,A -85,B 0,C 180,E1 -3320.476,E2 -3320.476} C_VEL
LIN {X 0,Y 552.069,Z 680.917,A -85,B 0,C 180,E1 -3321.397,E2 -3321.397} C_VEL
LIN {X 0,Y 551.949,Z 687.938,A -85,B 0,C 180,E1 -3322.317,E2 -3322.317} C_VEL
LIN {X 0,Y 551.824,Z 694.865,A -85,B 0,C 180,E1 -3323.418,E2 -3323.418} C_VEL
LIN {X 0,Y 551.802,Z 700.386,A -85,B 0,C 180,E1 -3324.519,E2 -3324.519} C_VEL
LIN {X 0,Y 551.764,Z 704.696,A -85,B 0,C 180,E1 -3325.617,E2 -3325.617} C_VEL
LIN {X 0,Y 551.724,Z 708.755,A -85,B 0,C 180,E1 -3327.079,E2 -3327.079} C_VEL
LIN {X 0,Y 551.657,Z 710.212,A -85,B 0,C 180,E1 -3327.81,E2 -3327.81} C_VEL
LIN {X 0,Y 551.641,Z 711.752,A -85,B 0,C 180,E1 -3329.27,E2 -3329.27} C_VEL
LIN {X 0,Y 551.64,Z 712,A -85,B 0,C 180,E1 -3330,E2 -3330} C_VEL
LIN {X 0,Y 551.645,Z 711.162,A -85,B 0,C 180,E1 -3331.46,E2 -3331.46} C_VEL
LIN {X 0,Y 551.657,Z 710.212,A -85,B 0,C 180,E1 -3332.19,E2 -3332.19} C_VEL
LIN {X 0,Y 551.751,Z 706.923,A -85,B 0,C 180,E1 -3333.651,E2 -3333.651} C_VEL
LIN {X 0,Y 551.724,Z 703.322,A -85,B 0,C 180,E1 -3334.749,E2 -3334.749} C_VEL
LIN {X 0,Y 551.86,Z 698.626,A -85,B 0,C 180,E1 -3335.847,E2 -3335.847} C_VEL
LIN {X 0,Y 551.836,Z 693.779,A -85,B 0,C 180,E1 -3336.765,E2 -3336.765} C_VEL
LIN {X 0,Y 551.949,Z 687.938,A -85,B 0,C 180,E1 -3337.683,E2 -3337.683} C_VEL
LIN {X 0,Y 552.069,Z 680.917,A -85,B 0,C 180,E1 -3338.603,E2 -3338.603} C_VEL
LIN {X 0,Y 552.197,Z 672.444,A -85,B 0,C 180,E1 -3339.524,E2 -3339.524} C_VEL
LIN {X 0,Y 552.412,Z 663.203,A -85,B 0,C 180,E1 -3340.352,E2 -3340.352} C_VEL
LIN {X 0,Y 552.619,Z 652.331,A -85,B 0,C 180,E1 -3341.147,E2 -3341.147} C_VEL
LIN {X 0,Y 552.752,Z 640.319,A -85,B 0,C 180,E1 -3341.831,E2 -3341.831} C_VEL
LIN {X 0,Y 552.872,Z 629.845,A -85,B 0,C 180,E1 -3342.294,E2 -3342.294} C_VEL
LIN {X 0,Y 553.035,Z 618.685,A -85,B 0,C 180,E1 -3342.663,E2 -3342.663} C_VEL
LIN {X 0,Y 553.108,Z 607.552,A -85,B 0,C 180,E1 -3342.918,E2 -3342.918} C_VEL
LIN {X 0,Y 553.345,Z 541.294,A -85,B 0,C 180,E1 -3343.8,E2 -3343.8} C_VEL
LIN {X 0,Y 553.317,Z 507.907,A -85,B 0,C 180,E1 -3344.238,E2 -3344.238} C_VEL
LIN {X 0,Y 552.244,Z 501.424,A -85,B 0,C 180,E1 -3344.379,E2 -3344.379} C_VEL
LIN {X 0,Y 552.241,Z 494.994,A -85,B 0,C 180,E1 -3345.501,E2 -3345.501} C_VEL
LIN {X 0,Y 552.515,Z 478.427,A -85,B 0,C 180,E1 -3348.542,E2 -3348.542} C_VEL
LIN {X 0,Y 552.704,Z 463.779,A -85,B 0,C 180,E1 -3351.247,E2 -3351.247} C_VEL
LIN {X 0,Y 553.018,Z 448.145,A -85,B 0,C 180,E1 -3354.195,E2 -3354.195} C_VEL
LIN {X 0,Y 552.111,Z 442.28,A -85,B 0,C 180,E1 -3355.404,E2 -3355.404} C_VEL
LIN {X 0,Y 552.07,Z 442.217,A -85,B 0,C 180,E1 -3358.551,E2 -3358.551} C_VEL
LIN {X 0,Y 552.093,Z 442.211,A -85,B 0,C 180,E1 -3361.471,E2 -3361.471} C_VEL
LIN {X 0,Y 552.094,Z 442.218,A -85,B 0,C 180,E1 -3364.163,E2 -3364.163} C_VEL
LIN {X 0,Y 552.047,Z 442.215,A -85,B 0,C 180,E1 -3366.751,E2 -3366.751} C_VEL
LIN {X 0,Y 552.09,Z 442.211,A -85,B 0,C 180,E1 -3369.53,E2 -3369.53} C_VEL
LIN {X 0,Y 552.08,Z 442.215,A -85,B 0,C 180,E1 -3372.43,E2 -3372.43} C_VEL
LIN {X 0,Y 552.066,Z 442.213,A -85,B 0,C 180,E1 -3375.559,E2 -3375.559} C_VEL
LIN {X 0,Y 552.05,Z 442.216,A -85,B 0,C 180,E1 -3378.547,E2 -3378.547} C_VEL
LIN {X 0,Y 552.086,Z 442.209,A -85,B 0,C 180,E1 -3381.408,E2 -3381.408} C_VEL
LIN {X 0,Y 552.058,Z 442.214,A -85,B 0,C 180,E1 -3384.562,E2 -3384.562} C_VEL
LIN {X 0,Y 552.094,Z 442.206,A -85,B 0,C 180,E1 -3387.156,E2 -3387.156} C_VEL
LIN {X 0,Y 552.085,Z 442.217,A -85,B 0,C 180,E1 -3389.954,E2 -3389.954} C_VEL
LIN {X 0,Y 552.072,Z 442.206,A -85,B 0,C 180,E1 -3393.012,E2 -3393.012} C_VEL
LIN {X 0,Y 552.071,Z 442.217,A -85,B 0,C 180,E1 -3395.96,E2 -3395.96} C_VEL
LIN {X 0,Y 552.083,Z 442.214,A -85,B 0,C 180,E1 -3398.335,E2 -3398.335} C_VEL
LIN {X 0,Y 552.078,Z 442.206,A -85,B 0,C 180,E1 -3400.671,E2 -3400.671} C_VEL
LIN {X 0,Y 552.06,Z 442.213,A -85,B 0,C 180,E1 -3403.735,E2 -3403.735} C_VEL
LIN {X 0,Y 552.101,Z 442.215,A -85,B 0,C 180,E1 -3406.003,E2 -3406.003} C_VEL
LIN {X 0,Y 552.121,Z 442.201,A -85,B 0,C 180,E1 -3408.992,E2 -3408.992} C_VEL
LIN {X 0,Y 552.103,Z 442.208,A -85,B 0,C 180,E1 -3411.95,E2 -3411.95} C_VEL
LIN {X 0,Y 552.195,Z 442.196,A -85,B 0,C 180,E1 -3414.888,E2 -3414.888} C_VEL
LIN {X 0,Y 552.214,Z 442.198,A -85,B 0,C 180,E1 -3417.811,E2 -3417.811} C_VEL
LIN {X 0,Y 552.216,Z 442.196,A -85,B 0,C 180,E1 -3419.999,E2 -3419.999} C_VEL
LIN {X 0,Y 552.166,Z 442.198,A -85,B 0,C 180,E1 -3422.917,E2 -3422.917} C_VEL
LIN {X 0,Y 552.168,Z 442.205,A -85,B 0,C 180,E1 -3425.843,E2 -3425.843} C_VEL
LIN {X 0,Y 552.115,Z 442.202,A -85,B 0,C 180,E1 -3428.785,E2 -3428.785} C_VEL
LIN {X 0,Y 552.093,Z 442.208,A -85,B 0,C 180,E1 -3431.751,E2 -3431.751} C_VEL
LIN {X 0,Y 552.111,Z 442.207,A -85,B 0,C 180,E1 -3434.748,E2 -3434.748} C_VEL
LIN {X 0,Y 552.06,Z 442.216,A -85,B 0,C 180,E1 -3437.789,E2 -3437.789} C_VEL
LIN {X 0,Y 552.092,Z 442.213,A -85,B 0,C 180,E1 -3440.101,E2 -3440.101} C_VEL
LIN {X 0,Y 552.07,Z 442.215,A -85,B 0,C 180,E1 -3442.45,E2 -3442.45} C_VEL
LIN {X 0,Y 552.067,Z 442.212,A -85,B 0,C 180,E1 -3445.332,E2 -3445.332} C_VEL
LIN {X 0,Y 552.041,Z 442.22,A -85,B 0,C 180,E1 -3448.1,E2 -3448.1} C_VEL
LIN {X 0,Y 552.077,Z 442.213,A -85,B 0,C 180,E1 -3450.609,E2 -3450.609} C_VEL
LIN {X 0,Y 552.082,Z 442.209,A -85,B 0,C 180,E1 -3453.186,E2 -3453.186} C_VEL
LIN {X 0,Y 552.067,Z 442.213,A -85,B 0,C 180,E1 -3453.756,E2 -3453.756} C_VEL
LIN {X 0,Y 551.412,Z 442.299,A -85,B 0,C 180,E1 -3454.365,E2 -3454.365} C_VEL
LIN {X 0,Y 548.542,Z 442.657,A -85,B 0,C 180,E1 -3455.353,E2 -3455.353} C_VEL
LIN {X 0,Y 546.11,Z 442.962,A -85,B 0,C 180,E1 -3456.148,E2 -3456.148} C_VEL
LIN {X 0,Y 545.069,Z 443.085,A -85,B 0,C 180,E1 -3456.762,E2 -3456.762} C_VEL
LIN {X 0,Y 544.987,Z 443.094,A -85,B 0,C 180,E1 -3456.97,E2 -3456.97} C_VEL
LIN {X 0,Y 545.056,Z 443.085,A -85,B 0,C 180,E1 -3459.318,E2 -3459.318} C_VEL
LIN {X 0,Y 545.02,Z 443.098,A -85,B 0,C 180,E1 -3462.106,E2 -3462.106} C_VEL
LIN {X 0,Y 545.005,Z 443.09,A -85,B 0,C 180,E1 -3465.171,E2 -3465.171} C_VEL
LIN {X 0,Y 545.014,Z 443.088,A -85,B 0,C 180,E1 -3467.891,E2 -3467.891} C_VEL
LIN {X 0,Y 545.047,Z 443.086,A -85,B 0,C 180,E1 -3470.816,E2 -3470.816} C_VEL
LIN {X 0,Y 544.986,Z 443.097,A -85,B 0,C 180,E1 -3473.616,E2 -3473.616} C_VEL
LIN {X 0,Y 545.025,Z 443.093,A -85,B 0,C 180,E1 -3476.326,E2 -3476.326} C_VEL
LIN {X 0,Y 545.036,Z 443.088,A -85,B 0,C 180,E1 -3478.951,E2 -3478.951} C_VEL
LIN {X 0,Y 545.018,Z 443.089,A -85,B 0,C 180,E1 -3481.503,E2 -3481.503} C_VEL
LIN {X 0,Y 545.014,Z 443.094,A -85,B 0,C 180,E1 -3484.505,E2 -3484.505} C_VEL
LIN {X 0,Y 545.01,Z 443.092,A -85,B 0,C 180,E1 -3487.241,E2 -3487.241} C_VEL
LIN {X 0,Y 545.085,Z 443.086,A -85,B 0,C 180,E1 -3490.414,E2 -3490.414} C_VEL
LIN {X 0,Y 545.003,Z 443.096,A -85,B 0,C 180,E1 -3493.519,E2 -3493.519} C_VEL
LIN {X 0,Y 545.061,Z 443.093,A -85,B 0,C 180,E1 -3495.819,E2 -3495.819} C_VEL
LIN {X 0,Y 545.055,Z 443.087,A -85,B 0,C 180,E1 -3498.848,E2 -3498.848} C_VEL
LIN {X 0,Y 545.05,Z 443.095,A -85,B 0,C 180,E1 -3501.846,E2 -3501.846} C_VEL
LIN {X 0,Y 545.145,Z 443.076,A -85,B 0,C 180,E1 -3504.822,E2 -3504.822} C_VEL
LIN {X 0,Y 545.175,Z 443.078,A -85,B 0,C 180,E1 -3507.784,E2 -3507.784} C_VEL
LIN {X 0,Y 545.175,Z 443.08,A -85,B 0,C 180,E1 -3510,E2 -3510} C_VEL
LIN {X 0,Y 545.126,Z 443.078,A -85,B 0,C 180,E1 -3512.956,E2 -3512.956} C_VEL
LIN {X 0,Y 545.112,Z 443.088,A -85,B 0,C 180,E1 -3515.92,E2 -3515.92} C_VEL
LIN {X 0,Y 545.073,Z 443.085,A -85,B 0,C 180,E1 -3518.901,E2 -3518.901} C_VEL
LIN {X 0,Y 545.049,Z 443.095,A -85,B 0,C 180,E1 -3521.906,E2 -3521.906} C_VEL
LIN {X 0,Y 545.062,Z 443.086,A -85,B 0,C 180,E1 -3524.944,E2 -3524.944} C_VEL
LIN {X 0,Y 545.03,Z 443.098,A -85,B 0,C 180,E1 -3528.027,E2 -3528.027} C_VEL
LIN {X 0,Y 545.066,Z 443.089,A -85,B 0,C 180,E1 -3530.373,E2 -3530.373} C_VEL
LIN {X 0,Y 545.054,Z 443.09,A -85,B 0,C 180,E1 -3533.56,E2 -3533.56} C_VEL
LIN {X 0,Y 545.02,Z 443.099,A -85,B 0,C 180,E1 -3536.003,E2 -3536.003} C_VEL
LIN {X 0,Y 545.004,Z 443.089,A -85,B 0,C 180,E1 -3538.735,E2 -3538.735} C_VEL
LIN {X 0,Y 545.036,Z 443.088,A -85,B 0,C 180,E1 -3541.049,E2 -3541.049} C_VEL
LIN {X 0,Y 545.025,Z 443.093,A -85,B 0,C 180,E1 -3543.674,E2 -3543.674} C_VEL
LIN {X 0,Y 544.986,Z 443.097,A -85,B 0,C 180,E1 -3546.384,E2 -3546.384} C_VEL
LIN {X 0,Y 545.036,Z 443.089,A -85,B 0,C 180,E1 -3549.318,E2 -3549.318} C_VEL
LIN {X 0,Y 545.014,Z 443.088,A -85,B 0,C 180,E1 -3552.109,E2 -3552.109} C_VEL
LIN {X 0,Y 545.005,Z 443.09,A -85,B 0,C 180,E1 -3555.172,E2 -3555.172} C_VEL
LIN {X 0,Y 545.02,Z 443.098,A -85,B 0,C 180,E1 -3557.894,E2 -3557.894} C_VEL
LIN {X 0,Y 545.061,Z 443.084,A -85,B 0,C 180,E1 -3560.819,E2 -3560.819} C_VEL
LIN {X 0,Y 544.989,Z 443.098,A -85,B 0,C 180,E1 -3563.617,E2 -3563.617} C_VEL
LIN {X 0,Y 545.029,Z 443.091,A -85,B 0,C 180,E1 -3566.327,E2 -3566.327} C_VEL
LIN {X 0,Y 545.04,Z 443.087,A -85,B 0,C 180,E1 -3568.952,E2 -3568.952} C_VEL
LIN {X 0,Y 545.023,Z 443.09,A -85,B 0,C 180,E1 -3571.505,E2 -3571.505} C_VEL
LIN {X 0,Y 545.018,Z 443.091,A -85,B 0,C 180,E1 -3574.507,E2 -3574.507} C_VEL
LIN {X 0,Y 545.016,Z 443.091,A -85,B 0,C 180,E1 -3577.243,E2 -3577.243} C_VEL
LIN {X 0,Y 545.073,Z 443.081,A -85,B 0,C 180,E1 -3580.259,E2 -3580.259} C_VEL
LIN {X 0,Y 545.015,Z 443.089,A -85,B 0,C 180,E1 -3582.749,E2 -3582.749} C_VEL
LIN {X 0,Y 545.057,Z 443.093,A -85,B 0,C 180,E1 -3585.82,E2 -3585.82} C_VEL
LIN {X 0,Y 545.062,Z 443.079,A -85,B 0,C 180,E1 -3588.85,E2 -3588.85} C_VEL
LIN {X 0,Y 545.057,Z 443.088,A -85,B 0,C 180,E1 -3591.847,E2 -3591.847} C_VEL
LIN {X 0,Y 545.153,Z 443.073,A -85,B 0,C 180,E1 -3594.824,E2 -3594.824} C_VEL
LIN {X 0,Y 545.183,Z 443.075,A -85,B 0,C 180,E1 -3597.785,E2 -3597.785} C_VEL
LIN {X 0,Y 545.184,Z 443.071,A -85,B 0,C 180,E1 -3600.001,E2 -3600.001} C_VEL
LIN {X 0,Y 545.134,Z 443.074,A -85,B 0,C 180,E1 -3602.957,E2 -3602.957} C_VEL
LIN {X 0,Y 545.118,Z 443.085,A -85,B 0,C 180,E1 -3605.921,E2 -3605.921} C_VEL
LIN {X 0,Y 545.061,Z 443.077,A -85,B 0,C 180,E1 -3608.902,E2 -3608.902} C_VEL
LIN {X 0,Y 545.061,Z 443.09,A -85,B 0,C 180,E1 -3611.907,E2 -3611.907} C_VEL
LIN {X 0,Y 545.034,Z 443.087,A -85,B 0,C 180,E1 -3614.946,E2 -3614.946} C_VEL
LIN {X 0,Y 545.03,Z 443.089,A -85,B 0,C 180,E1 -3618.028,E2 -3618.028} C_VEL
LIN {X 0,Y 545.001,Z 443.093,A -85,B 0,C 180,E1 -3620.377,E2 -3620.377} C_VEL
LIN {X 0,Y 545.023,Z 443.089,A -85,B 0,C 180,E1 -3622.759,E2 -3622.759} C_VEL
LIN {X 0,Y 545.027,Z 443.09,A -85,B 0,C 180,E1 -3625.495,E2 -3625.495} C_VEL
LIN {X 0,Y 545.029,Z 443.089,A -85,B 0,C 180,E1 -3628.497,E2 -3628.497} C_VEL
LIN {X 0,Y 545.051,Z 443.086,A -85,B 0,C 180,E1 -3631.05,E2 -3631.05} C_VEL
LIN {X 0,Y 545.039,Z 443.091,A -85,B 0,C 180,E1 -3633.675,E2 -3633.675} C_VEL
LIN {X 0,Y 545,Z 443.095,A -85,B 0,C 180,E1 -3636.384,E2 -3636.384} C_VEL
LIN {X 0,Y 545.032,Z 443.088,A -85,B 0,C 180,E1 -3639.315,E2 -3639.315} C_VEL
LIN {X 0,Y 545.027,Z 443.095,A -85,B 0,C 180,E1 -3642.109,E2 -3642.109} C_VEL
LIN {X 0,Y 545.017,Z 443.09,A -85,B 0,C 180,E1 -3645.173,E2 -3645.173} C_VEL
LIN {X 0,Y 545.029,Z 443.094,A -85,B 0,C 180,E1 -3647.893,E2 -3647.893} C_VEL
LIN {X 0,Y 545.062,Z 443.084,A -85,B 0,C 180,E1 -3650.817,E2 -3650.817} C_VEL
LIN {X 0,Y 544.999,Z 443.097,A -85,B 0,C 180,E1 -3653.617,E2 -3653.617} C_VEL
LIN {X 0,Y 545.035,Z 443.09,A -85,B 0,C 180,E1 -3656.326,E2 -3656.326} C_VEL
LIN {X 0,Y 545.04,Z 443.089,A -85,B 0,C 180,E1 -3658.951,E2 -3658.951} C_VEL
LIN {X 0,Y 545.031,Z 443.095,A -85,B 0,C 180,E1 -3661.504,E2 -3661.504} C_VEL
LIN {X 0,Y 545.091,Z 443.294,A -85,B 0,C 180,E1 -3664.493,E2 -3664.493} C_VEL
LIN {X 0,Y 546.042,Z 449.063,A -85,B 0,C 180,E1 -3665.678,E2 -3665.678} C_VEL
LIN {X 0,Y 545.741,Z 463.641,A -85,B 0,C 180,E1 -3668.468,E2 -3668.468} C_VEL
LIN {X 0,Y 545.535,Z 477.245,A -85,B 0,C 180,E1 -3671.017,E2 -3671.017} C_VEL
LIN {X 0,Y 545.285,Z 491.872,A -85,B 0,C 180,E1 -3673.72,E2 -3673.72} C_VEL
LIN {X 0,Y 545.194,Z 501.251,A -85,B 0,C 180,E1 -3675.416,E2 -3675.416} C_VEL
LIN {X 0,Y 545.602,Z 503.792,A -85,B 0,C 180,E1 -3675.501,E2 -3675.501} C_VEL
LIN {X 0,Y 546.535,Z 510.733,A -85,B 0,C 180,E1 -3675.619,E2 -3675.619} C_VEL
LIN {X 0,Y 546.186,Z 606.18,A -85,B 0,C 180,E1 -3676.892,E2 -3676.892} C_VEL
LIN {X 0,Y 546.145,Z 616.933,A -85,B 0,C 180,E1 -3677.128,E2 -3677.128} C_VEL
LIN {X 0,Y 545.981,Z 627.301,A -85,B 0,C 180,E1 -3677.454,E2 -3677.454} C_VEL
LIN {X 0,Y 545.849,Z 636.374,A -85,B 0,C 180,E1 -3677.829,E2 -3677.829} C_VEL
LIN {X 0,Y 545.728,Z 646.249,A -85,B 0,C 180,E1 -3678.342,E2 -3678.342} C_VEL
LIN {X 0,Y 545.545,Z 655.797,A -85,B 0,C 180,E1 -3678.952,E2 -3678.952} C_VEL
LIN {X 0,Y 545.369,Z 664.286,A -85,B 0,C 180,E1 -3679.606,E2 -3679.606} C_VEL
LIN {X 0,Y 545.163,Z 672.433,A -85,B 0,C 180,E1 -3680.352,E2 -3680.352} C_VEL
LIN {X 0,Y 545.028,Z 679.352,A -85,B 0,C 180,E1 -3681.099,E2 -3681.099} C_VEL
LIN {X 0,Y 544.917,Z 686.622,A -85,B 0,C 180,E1 -3682.031,E2 -3682.031} C_VEL
LIN {X 0,Y 544.791,Z 692.683,A -85,B 0,C 180,E1 -3682.961,E2 -3682.961} C_VEL
LIN {X 0,Y 544.724,Z 696.647,A -85,B 0,C 180,E1 -3683.665,E2 -3683.665} C_VEL
LIN {X 0,Y 544.653,Z 701.898,A -85,B 0,C 180,E1 -3684.818,E2 -3684.818} C_VEL
LIN {X 0,Y 544.684,Z 705.836,A -85,B 0,C 180,E1 -3685.931,E2 -3685.931} C_VEL
LIN {X 0,Y 544.651,Z 708.748,A -85,B 0,C 180,E1 -3687.041,E2 -3687.041} C_VEL
LIN {X 0,Y 544.571,Z 710.213,A -85,B 0,C 180,E1 -3687.781,E2 -3687.781} C_VEL
LIN {X 0,Y 544.542,Z 711.744,A -85,B 0,C 180,E1 -3689.261,E2 -3689.261} C_VEL
LIN {X 0,Y 544.541,Z 712,A -85,B 0,C 180,E1 -3690,E2 -3690} C_VEL
LIN {X 0,Y 544.546,Z 711.155,A -85,B 0,C 180,E1 -3691.479,E2 -3691.479} C_VEL
LIN {X 0,Y 544.571,Z 710.213,A -85,B 0,C 180,E1 -3692.219,E2 -3692.219} C_VEL
LIN {X 0,Y 544.669,Z 706.916,A -85,B 0,C 180,E1 -3693.699,E2 -3693.699} C_VEL
LIN {X 0,Y 544.628,Z 703.316,A -85,B 0,C 180,E1 -3694.811,E2 -3694.811} C_VEL
LIN {X 0,Y 544.769,Z 698.619,A -85,B 0,C 180,E1 -3695.924,E2 -3695.924} C_VEL
LIN {X 0,Y 544.786,Z 693.77,A -85,B 0,C 180,E1 -3696.853,E2 -3696.853} C_VEL
LIN {X 0,Y 544.896,Z 687.928,A -85,B 0,C 180,E1 -3697.783,E2 -3697.783} C_VEL
LIN {X 0,Y 545.02,Z 680.907,A -85,B 0,C 180,E1 -3698.715,E2 -3698.715} C_VEL
LIN {X 0,Y 545.136,Z 674.277,A -85,B 0,C 180,E1 -3699.461,E2 -3699.461} C_VEL
LIN {X 0,Y 545.312,Z 665.381,A -85,B 0,C 180,E1 -3700.301,E2 -3700.301} C_VEL
LIN {X 0,Y 545.514,Z 657.107,A -85,B 0,C 180,E1 -3700.954,E2 -3700.954} C_VEL
LIN {X 0,Y 545.669,Z 648.33,A -85,B 0,C 180,E1 -3701.536,E2 -3701.536} C_VEL
LIN {X 0,Y 545.797,Z 640.305,A -85,B 0,C 180,E1 -3701.984,E2 -3701.984} C_VEL
LIN {X 0,Y 545.923,Z 629.823,A -85,B 0,C 180,E1 -3702.453,E2 -3702.453} C_VEL
LIN {X 0,Y 546.115,Z 618.653,A -85,B 0,C 180,E1 -3702.826,E2 -3702.826} C_VEL
LIN {X 0,Y 546.193,Z 608.823,A -85,B 0,C 180,E1 -3703.06,E2 -3703.06} C_VEL
LIN {X 0,Y 546.341,Z 586.011,A -85,B 0,C 180,E1 -3703.388,E2 -3703.388} C_VEL
LIN {X 0,Y 546.408,Z 508.401,A -85,B 0,C 180,E1 -3704.416,E2 -3704.416} C_VEL
LIN {X 0,Y 545.206,Z 501.48,A -85,B 0,C 180,E1 -3704.565,E2 -3704.565} C_VEL
LIN {X 0,Y 545.219,Z 497.064,A -85,B 0,C 180,E1 -3705.322,E2 -3705.322} C_VEL
LIN {X 0,Y 545.489,Z 480.382,A -85,B 0,C 180,E1 -3708.4,E2 -3708.4} C_VEL
LIN {X 0,Y 545.734,Z 465.736,A -85,B 0,C 180,E1 -3711.136,E2 -3711.136} C_VEL
LIN {X 0,Y 546.023,Z 450.985,A -85,B 0,C 180,E1 -3713.955,E2 -3713.955} C_VEL
LIN {X 0,Y 545.79,Z 447.003,A -85,B 0,C 180,E1 -3714.739,E2 -3714.739} C_VEL
LIN {X 0,Y 545.065,Z 443.162,A -85,B 0,C 180,E1 -3715.566,E2 -3715.566} C_VEL
LIN {X 0,Y 545.018,Z 443.094,A -85,B 0,C 180,E1 -3718.733,E2 -3718.733} C_VEL
LIN {X 0,Y 545.04,Z 443.089,A -85,B 0,C 180,E1 -3721.049,E2 -3721.049} C_VEL
LIN {X 0,Y 545.051,Z 443.088,A -85,B 0,C 180,E1 -3723.672,E2 -3723.672} C_VEL
LIN {X 0,Y 544.999,Z 443.097,A -85,B 0,C 180,E1 -3726.383,E2 -3726.383} C_VEL
LIN {X 0,Y 545.05,Z 443.086,A -85,B 0,C 180,E1 -3729.316,E2 -3729.316} C_VEL
LIN {X 0,Y 545.029,Z 443.093,A -85,B 0,C 180,E1 -3732.107,E2 -3732.107} C_VEL
LIN {X 0,Y 545.015,Z 443.09,A -85,B 0,C 180,E1 -3735.171,E2 -3735.171} C_VEL
LIN {X 0,Y 545.019,Z 443.094,A -85,B 0,C 180,E1 -3738.409,E2 -3738.409} C_VEL
LIN {X 0,Y 545.041,Z 443.086,A -85,B 0,C 180,E1 -3740.814,E2 -3740.814} C_VEL
LIN {X 0,Y 545,Z 443.095,A -85,B 0,C 180,E1 -3743.616,E2 -3743.616} C_VEL
LIN {X 0,Y 545.039,Z 443.091,A -85,B 0,C 180,E1 -3746.325,E2 -3746.325} C_VEL
LIN {X 0,Y 545.051,Z 443.086,A -85,B 0,C 180,E1 -3748.95,E2 -3748.95} C_VEL
LIN {X 0,Y 545.029,Z 443.089,A -85,B 0,C 180,E1 -3751.503,E2 -3751.503} C_VEL
LIN {X 0,Y 545.027,Z 443.09,A -85,B 0,C 180,E1 -3754.505,E2 -3754.505} C_VEL
LIN {X 0,Y 545.023,Z 443.089,A -85,B 0,C 180,E1 -3757.241,E2 -3757.241} C_VEL
LIN {X 0,Y 545.001,Z 443.093,A -85,B 0,C 180,E1 -3759.623,E2 -3759.623} C_VEL
LIN {X 0,Y 545.02,Z 443.087,A -85,B 0,C 180,E1 -3762.747,E2 -3762.747} C_VEL
LIN {X 0,Y 545.06,Z 443.089,A -85,B 0,C 180,E1 -3765.818,E2 -3765.818} C_VEL
LIN {X 0,Y 545.066,Z 443.08,A -85,B 0,C 180,E1 -3768.847,E2 -3768.847} C_VEL
LIN {X 0,Y 545.06,Z 443.083,A -85,B 0,C 180,E1 -3771.845,E2 -3771.845} C_VEL
LIN {X 0,Y 545.154,Z 443.073,A -85,B 0,C 180,E1 -3774.821,E2 -3774.821} C_VEL
LIN {X 0,Y 545.185,Z 443.073,A -85,B 0,C 180,E1 -3777.783,E2 -3777.783} C_VEL
LIN {X 0,Y 545.184,Z 443.071,A -85,B 0,C 180,E1 -3779.999,E2 -3779.999} C_VEL
LIN {X 0,Y 545.134,Z 443.073,A -85,B 0,C 180,E1 -3782.955,E2 -3782.955} C_VEL
LIN {X 0,Y 545.119,Z 443.085,A -85,B 0,C 180,E1 -3785.919,E2 -3785.919} C_VEL
LIN {X 0,Y 545.058,Z 443.08,A -85,B 0,C 180,E1 -3788.9,E2 -3788.9} C_VEL
LIN {X 0,Y 545.058,Z 443.087,A -85,B 0,C 180,E1 -3791.905,E2 -3791.905} C_VEL
LIN {X 0,Y 545.066,Z 443.084,A -85,B 0,C 180,E1 -3794.943,E2 -3794.943} C_VEL
LIN {X 0,Y 545.026,Z 443.093,A -85,B 0,C 180,E1 -3798.026,E2 -3798.026} C_VEL
LIN {X 0,Y 545.033,Z 443.09,A -85,B 0,C 180,E1 -3800.373,E2 -3800.373} C_VEL
LIN {X 0,Y 545.016,Z 443.091,A -85,B 0,C 180,E1 -3802.757,E2 -3802.757} C_VEL
LIN {X 0,Y 545.017,Z 443.091,A -85,B 0,C 180,E1 -3805.493,E2 -3805.493} C_VEL
LIN {X 0,Y 545.023,Z 443.09,A -85,B 0,C 180,E1 -3808.495,E2 -3808.495} C_VEL
LIN {X 0,Y 545.04,Z 443.087,A -85,B 0,C 180,E1 -3811.048,E2 -3811.048} C_VEL
LIN {X 0,Y 545.025,Z 443.091,A -85,B 0,C 180,E1 -3813.753,E2 -3813.753} C_VEL
LIN {X 0,Y 544.989,Z 443.098,A -85,B 0,C 180,E1 -3816.383,E2 -3816.383} C_VEL
LIN {X 0,Y 544.987,Z 443.094,A -85,B 0,C 180,E1 -3816.97,E2 -3816.97} C_VEL
LIN {X 0,Y 544.33,Z 443.18,A -85,B 0,C 180,E1 -3817.587,E2 -3817.587} C_VEL
LIN {X 0,Y 541.49,Z 443.533,A -85,B 0,C 180,E1 -3818.589,E2 -3818.589} C_VEL
LIN {X 0,Y 539.085,Z 443.833,A -85,B 0,C 180,E1 -3819.395,E2 -3819.395} C_VEL
LIN {X 0,Y 538.054,Z 443.963,A -85,B 0,C 180,E1 -3820.018,E2 -3820.018} C_VEL
LIN {X 0,Y 537.971,Z 443.967,A -85,B 0,C 180,E1 -3820.228,E2 -3820.228} C_VEL
LIN {X 0,Y 537.955,Z 443.97,A -85,B 0,C 180,E1 -3822.98,E2 -3822.98} C_VEL
LIN {X 0,Y 537.984,Z 443.97,A -85,B 0,C 180,E1 -3825.928,E2 -3825.928} C_VEL
LIN {X 0,Y 537.964,Z 443.966,A -85,B 0,C 180,E1 -3828.221,E2 -3828.221} C_VEL
LIN {X 0,Y 537.984,Z 443.966,A -85,B 0,C 180,E1 -3831.168,E2 -3831.168} C_VEL
LIN {X 0,Y 537.942,Z 443.974,A -85,B 0,C 180,E1 -3834.093,E2 -3834.093} C_VEL
LIN {X 0,Y 537.998,Z 443.964,A -85,B 0,C 180,E1 -3836.726,E2 -3836.726} C_VEL
LIN {X 0,Y 537.985,Z 443.969,A -85,B 0,C 180,E1 -3839.56,E2 -3839.56} C_VEL
LIN {X 0,Y 537.974,Z 443.97,A -85,B 0,C 180,E1 -3842.661,E2 -3842.661} C_VEL
LIN {X 0,Y 537.961,Z 443.971,A -85,B 0,C 180,E1 -3845.289,E2 -3845.289} C_VEL
LIN {X 0,Y 537.997,Z 443.974,A -85,B 0,C 180,E1 -3848.042,E2 -3848.042} C_VEL
LIN {X 0,Y 537.989,Z 443.967,A -85,B 0,C 180,E1 -3850.938,E2 -3850.938} C_VEL
LIN {X 0,Y 537.951,Z 443.973,A -85,B 0,C 180,E1 -3853.297,E2 -3853.297} C_VEL
LIN {X 0,Y 538.031,Z 443.966,A -85,B 0,C 180,E1 -3855.63,E2 -3855.63} C_VEL
LIN {X 0,Y 538.007,Z 443.966,A -85,B 0,C 180,E1 -3858.7,E2 -3858.7} C_VEL
LIN {X 0,Y 538.021,Z 443.969,A -85,B 0,C 180,E1 -3861.739,E2 -3861.739} C_VEL
LIN {X 0,Y 538.105,Z 443.954,A -85,B 0,C 180,E1 -3864.754,E2 -3864.754} C_VEL
LIN {X 0,Y 538.146,Z 443.953,A -85,B 0,C 180,E1 -3867.755,E2 -3867.755} C_VEL
LIN {X 0,Y 538.143,Z 443.956,A -85,B 0,C 180,E1 -3870,E2 -3870} C_VEL
LIN {X 0,Y 538.093,Z 443.954,A -85,B 0,C 180,E1 -3872.995,E2 -3872.995} C_VEL
LIN {X 0,Y 538.069,Z 443.965,A -85,B 0,C 180,E1 -3875.998,E2 -3875.998} C_VEL
LIN {X 0,Y 538.026,Z 443.963,A -85,B 0,C 180,E1 -3879.018,E2 -3879.018} C_VEL
LIN {X 0,Y 538.02,Z 443.971,A -85,B 0,C 180,E1 -3882.064,E2 -3882.064} C_VEL
LIN {X 0,Y 538.02,Z 443.963,A -85,B 0,C 180,E1 -3885.144,E2 -3885.144} C_VEL
LIN {X 0,Y 537.985,Z 443.973,A -85,B 0,C 180,E1 -3888.272,E2 -3888.272} C_VEL
LIN {X 0,Y 538.008,Z 443.965,A -85,B 0,C 180,E1 -3890.652,E2 -3890.652} C_VEL
LIN {X 0,Y 537.989,Z 443.967,A -85,B 0,C 180,E1 -3893.073,E2 -3893.073} C_VEL
LIN {X 0,Y 537.973,Z 443.973,A -85,B 0,C 180,E1 -3895.661,E2 -3895.661} C_VEL
LIN {X 0,Y 537.957,Z 443.975,A -85,B 0,C 180,E1 -3898.054,E2 -3898.054} C_VEL
LIN {X 0,Y 537.985,Z 443.967,A -85,B 0,C 180,E1 -3900.629,E2 -3900.629} C_VEL
LIN {X 0,Y 538.004,Z 443.964,A -85,B 0,C 180,E1 -3903.279,E2 -3903.279} C_VEL
LIN {X 0,Y 537.939,Z 443.976,A -85,B 0,C 180,E1 -3906.008,E2 -3906.008} C_VEL
LIN {X 0,Y 537.984,Z 443.966,A -85,B 0,C 180,E1 -3908.832,E2 -3908.832} C_VEL
LIN {X 0,Y 537.96,Z 443.966,A -85,B 0,C 180,E1 -3911.873,E2 -3911.873} C_VEL
LIN {X 0,Y 537.978,Z 443.965,A -85,B 0,C 180,E1 -3914.865,E2 -3914.865} C_VEL
LIN {X 0,Y 537.956,Z 443.97,A -85,B 0,C 180,E1 -3917.21,E2 -3917.21} C_VEL
LIN {X 0,Y 537.991,Z 443.971,A -85,B 0,C 180,E1 -3920.202,E2 -3920.202} C_VEL
LIN {X 0,Y 537.942,Z 443.971,A -85,B 0,C 180,E1 -3923.063,E2 -3923.063} C_VEL
LIN {X 0,Y 537.982,Z 443.969,A -85,B 0,C 180,E1 -3925.826,E2 -3925.826} C_VEL
LIN {X 0,Y 537.982,Z 443.969,A -85,B 0,C 180,E1 -3928.499,E2 -3928.499} C_VEL
LIN {X 0,Y 537.972,Z 443.966,A -85,B 0,C 180,E1 -3931.096,E2 -3931.096} C_VEL
LIN {X 0,Y 537.967,Z 443.967,A -85,B 0,C 180,E1 -3933.631,E2 -3933.631} C_VEL
LIN {X 0,Y 537.996,Z 443.971,A -85,B 0,C 180,E1 -3936.124,E2 -3936.124} C_VEL
LIN {X 0,Y 537.998,Z 443.963,A -85,B 0,C 180,E1 -3938.546,E2 -3938.546} C_VEL
LIN {X 0,Y 537.964,Z 443.961,A -85,B 0,C 180,E1 -3940.939,E2 -3940.939} C_VEL
LIN {X 0,Y 537.955,Z 443.969,A -85,B 0,C 180,E1 -3943.298,E2 -3943.298} C_VEL
LIN {X 0,Y 538.03,Z 443.965,A -85,B 0,C 180,E1 -3945.631,E2 -3945.631} C_VEL
LIN {X 0,Y 538.014,Z 443.957,A -85,B 0,C 180,E1 -3948.702,E2 -3948.702} C_VEL
LIN {X 0,Y 538.026,Z 443.962,A -85,B 0,C 180,E1 -3951.74,E2 -3951.74} C_VEL
LIN {X 0,Y 538.113,Z 443.95,A -85,B 0,C 180,E1 -3954.756,E2 -3954.756} C_VEL
LIN {X 0,Y 538.154,Z 443.95,A -85,B 0,C 180,E1 -3957.756,E2 -3957.756} C_VEL
LIN {X 0,Y 538.153,Z 443.946,A -85,B 0,C 180,E1 -3960.001,E2 -3960.001} C_VEL
LIN {X 0,Y 538.102,Z 443.95,A -85,B 0,C 180,E1 -3962.996,E2 -3962.996} C_VEL
LIN {X 0,Y 538.074,Z 443.961,A -85,B 0,C 180,E1 -3965.999,E2 -3965.999} C_VEL
LIN {X 0,Y 538.019,Z 443.954,A -85,B 0,C 180,E1 -3969.02,E2 -3969.02} C_VEL
LIN {X 0,Y 538.032,Z 443.966,A -85,B 0,C 180,E1 -3972.065,E2 -3972.065} C_VEL
LIN {X 0,Y 537.982,Z 443.966,A -85,B 0,C 180,E1 -3975.147,E2 -3975.147} C_VEL
LIN {X 0,Y 537.979,Z 443.964,A -85,B 0,C 180,E1 -3978.273,E2 -3978.273} C_VEL
LIN {X 0,Y 537.969,Z 443.967,A -85,B 0,C 180,E1 -3980.655,E2 -3980.655} C_VEL
LIN {X 0,Y 538.003,Z 443.963,A -85,B 0,C 180,E1 -3983.073,E2 -3983.073} C_VEL
LIN {X 0,Y 537.986,Z 443.969,A -85,B 0,C 180,E1 -3985.661,E2 -3985.661} C_VEL
LIN {X 0,Y 537.968,Z 443.974,A -85,B 0,C 180,E1 -3988.055,E2 -3988.055} C_VEL
LIN {X 0,Y 537.999,Z 443.965,A -85,B 0,C 180,E1 -3990.629,E2 -3990.629} C_VEL
LIN {X 0,Y 538.019,Z 443.96,A -85,B 0,C 180,E1 -3993.279,E2 -3993.279} C_VEL
LIN {X 0,Y 537.953,Z 443.978,A -85,B 0,C 180,E1 -3996.009,E2 -3996.009} C_VEL
LIN {X 0,Y 537.983,Z 443.965,A -85,B 0,C 180,E1 -3998.834,E2 -3998.834} C_VEL
LIN {X 0,Y 537.974,Z 443.976,A -85,B 0,C 180,E1 -4001.873,E2 -4001.873} C_VEL
LIN {X 0,Y 537.989,Z 443.965,A -85,B 0,C 180,E1 -4004.865,E2 -4004.865} C_VEL
LIN {X 0,Y 537.969,Z 443.969,A -85,B 0,C 180,E1 -4007.21,E2 -4007.21} C_VEL
LIN {X 0,Y 537.988,Z 443.968,A -85,B 0,C 180,E1 -4010.422,E2 -4010.422} C_VEL
LIN {X 0,Y 537.953,Z 443.97,A -85,B 0,C 180,E1 -4013.062,E2 -4013.062} C_VEL
LIN {X 0,Y 537.991,Z 443.974,A -85,B 0,C 180,E1 -4015.825,E2 -4015.825} C_VEL
LIN {X 0,Y 537.992,Z 443.969,A -85,B 0,C 180,E1 -4018.498,E2 -4018.498} C_VEL
LIN {X 0,Y 537.986,Z 443.969,A -85,B 0,C 180,E1 -4021.096,E2 -4021.096} C_VEL
LIN {X 0,Y 538.045,Z 444.082,A -85,B 0,C 180,E1 -4024.299,E2 -4024.299} C_VEL
LIN {X 0,Y 539.104,Z 450.569,A -85,B 0,C 180,E1 -4025.661,E2 -4025.661} C_VEL
LIN {X 0,Y 538.739,Z 465.597,A -85,B 0,C 180,E1 -4028.576,E2 -4028.576} C_VEL
LIN {X 0,Y 538.48,Z 480.245,A -85,B 0,C 180,E1 -4031.352,E2 -4031.352} C_VEL
LIN {X 0,Y 538.181,Z 495.912,A -85,B 0,C 180,E1 -4034.278,E2 -4034.278} C_VEL
LIN {X 0,Y 538.174,Z 501.309,A -85,B 0,C 180,E1 -4035.235,E2 -4035.235} C_VEL
LIN {X 0,Y 539.138,Z 506.981,A -85,B 0,C 180,E1 -4035.367,E2 -4035.367} C_VEL
LIN {X 0,Y 539.674,Z 512.454,A -85,B 0,C 180,E1 -4035.456,E2 -4035.456} C_VEL
LIN {X 0,Y 539.283,Z 606.129,A -85,B 0,C 180,E1 -4036.721,E2 -4036.721} C_VEL
LIN {X 0,Y 539.259,Z 616.04,A -85,B 0,C 180,E1 -4036.936,E2 -4036.936} C_VEL
LIN {X 0,Y 539.1,Z 626.018,A -85,B 0,C 180,E1 -4037.244,E2 -4037.244} C_VEL
LIN {X 0,Y 538.894,Z 636.359,A -85,B 0,C 180,E1 -4037.669,E2 -4037.669} C_VEL
LIN {X 0,Y 538.748,Z 646.235,A -85,B 0,C 180,E1 -4038.189,E2 -4038.189} C_VEL
LIN {X 0,Y 538.61,Z 654.473,A -85,B 0,C 180,E1 -4038.713,E2 -4038.713} C_VEL
LIN {X 0,Y 538.414,Z 663.178,A -85,B 0,C 180,E1 -4039.375,E2 -4039.375} C_VEL
LIN {X 0,Y 538.217,Z 670.577,A -85,B 0,C 180,E1 -4040.037,E2 -4040.037} C_VEL
LIN {X 0,Y 537.983,Z 679.341,A -85,B 0,C 180,E1 -4040.981,E2 -4040.981} C_VEL
LIN {X 0,Y 537.851,Z 686.613,A -85,B 0,C 180,E1 -4041.925,E2 -4041.925} C_VEL
LIN {X 0,Y 537.733,Z 692.674,A -85,B 0,C 180,E1 -4042.868,E2 -4042.868} C_VEL
LIN {X 0,Y 537.636,Z 697.115,A -85,B 0,C 180,E1 -4043.681,E2 -4043.681} C_VEL
LIN {X 0,Y 537.587,Z 701.892,A -85,B 0,C 180,E1 -4044.749,E2 -4044.749} C_VEL
LIN {X 0,Y 537.604,Z 705.829,A -85,B 0,C 180,E1 -4045.877,E2 -4045.877} C_VEL
LIN {X 0,Y 537.551,Z 708.741,A -85,B 0,C 180,E1 -4047.002,E2 -4047.002} C_VEL
LIN {X 0,Y 537.49,Z 710.214,A -85,B 0,C 180,E1 -4047.752,E2 -4047.752} C_VEL
LIN {X 0,Y 537.442,Z 711.737,A -85,B 0,C 180,E1 -4049.251,E2 -4049.251} C_VEL
LIN {X 0,Y 537.442,Z 712,A -85,B 0,C 180,E1 -4050,E2 -4050} C_VEL
LIN {X 0,Y 537.451,Z 711.147,A -85,B 0,C 180,E1 -4051.499,E2 -4051.499} C_VEL
LIN {X 0,Y 537.49,Z 710.214,A -85,B 0,C 180,E1 -4052.248,E2 -4052.248} C_VEL
LIN {X 0,Y 537.591,Z 706.909,A -85,B 0,C 180,E1 -4053.748,E2 -4053.748} C_VEL
LIN {X 0,Y 537.54,Z 703.31,A -85,B 0,C 180,E1 -4054.875,E2 -4054.875} C_VEL
LIN {X 0,Y 537.679,Z 698.611,A -85,B 0,C 180,E1 -4056.002,E2 -4056.002} C_VEL
LIN {X 0,Y 537.729,Z 693.761,A -85,B 0,C 180,E1 -4056.944,E2 -4056.944} C_VEL
LIN {X 0,Y 537.83,Z 687.919,A -85,B 0,C 180,E1 -4057.886,E2 -4057.886} C_VEL
LIN {X 0,Y 537.965,Z 682.451,A -85,B 0,C 180,E1 -4058.641,E2 -4058.641} C_VEL
LIN {X 0,Y 538.113,Z 674.266,A -85,B 0,C 180,E1 -4059.585,E2 -4059.585} C_VEL
LIN {X 0,Y 538.269,Z 666.464,A -85,B 0,C 180,E1 -4060.342,E2 -4060.342} C_VEL
LIN {X 0,Y 538.511,Z 658.403,A -85,B 0,C 180,E1 -4061.003,E2 -4061.003} C_VEL
LIN {X 0,Y 538.687,Z 648.999,A -85,B 0,C 180,E1 -4061.647,E2 -4061.647} C_VEL
LIN {X 0,Y 538.835,Z 640.29,A -85,B 0,C 180,E1 -4062.141,E2 -4062.141} C_VEL
LIN {X 0,Y 538.999,Z 629.801,A -85,B 0,C 180,E1 -4062.615,E2 -4062.615} C_VEL
LIN {X 0,Y 539.203,Z 619.482,A -85,B 0,C 180,E1 -4062.969,E2 -4062.969} C_VEL
LIN {X 0,Y 539.286,Z 608.772,A -85,B 0,C 180,E1 -4063.231,E2 -4063.231} C_VEL
LIN {X 0,Y 539.423,Z 587.797,A -85,B 0,C 180,E1 -4063.539,E2 -4063.539} C_VEL
LIN {X 0,Y 539.508,Z 508.965,A -85,B 0,C 180,E1 -4064.596,E2 -4064.596} C_VEL
LIN {X 0,Y 538.204,Z 501.69,A -85,B 0,C 180,E1 -4064.742,E2 -4064.742} C_VEL
LIN {X 0,Y 538.147,Z 500.381,A -85,B 0,C 180,E1 -4064.891,E2 -4064.891} C_VEL
LIN {X 0,Y 538.5,Z 482.337,A -85,B 0,C 180,E1 -4068.253,E2 -4068.253} C_VEL
LIN {X 0,Y 538.748,Z 466.652,A -85,B 0,C 180,E1 -4071.223,E2 -4071.223} C_VEL
LIN {X 0,Y 539.07,Z 451.667,A -85,B 0,C 180,E1 -4074.13,E2 -4074.13} C_VEL
LIN {X 0,Y 538.551,Z 446.902,A -85,B 0,C 180,E1 -4075.095,E2 -4075.095} C_VEL
LIN {X 0,Y 538.019,Z 444.047,A -85,B 0,C 180,E1 -4075.729,E2 -4075.729} C_VEL
LIN {X 0,Y 537.986,Z 443.969,A -85,B 0,C 180,E1 -4078.904,E2 -4078.904} C_VEL
LIN {X 0,Y 537.996,Z 443.973,A -85,B 0,C 180,E1 -4081.884,E2 -4081.884} C_VEL
LIN {X 0,Y 537.994,Z 443.968,A -85,B 0,C 180,E1 -4084.614,E2 -4084.614} C_VEL
LIN {X 0,Y 537.978,Z 443.972,A -85,B 0,C 180,E1 -4087.878,E2 -4087.878} C_VEL
LIN {X 0,Y 537.952,Z 443.965,A -85,B 0,C 180,E1 -4090.784,E2 -4090.784} C_VEL
LIN {X 0,Y 537.979,Z 443.972,A -85,B 0,C 180,E1 -4093.818,E2 -4093.818} C_VEL
LIN {X 0,Y 537.977,Z 443.974,A -85,B 0,C 180,E1 -4096.18,E2 -4096.18} C_VEL
LIN {X 0,Y 537.951,Z 443.97,A -85,B 0,C 180,E1 -4099.264,E2 -4099.264} C_VEL
LIN {X 0,Y 537.97,Z 443.977,A -85,B 0,C 180,E1 -4102.12,E2 -4102.12} C_VEL
LIN {X 0,Y 537.992,Z 443.963,A -85,B 0,C 180,E1 -4105.385,E2 -4105.385} C_VEL
LIN {X 0,Y 537.995,Z 443.972,A -85,B 0,C 180,E1 -4108.115,E2 -4108.115} C_VEL
LIN {X 0,Y 537.982,Z 443.965,A -85,B 0,C 180,E1 -4111.094,E2 -4111.094} C_VEL
LIN {X 0,Y 537.976,Z 443.964,A -85,B 0,C 180,E1 -4113.629,E2 -4113.629} C_VEL
LIN {X 0,Y 538.004,Z 443.972,A -85,B 0,C 180,E1 -4116.122,E2 -4116.122} C_VEL
LIN {X 0,Y 537.995,Z 443.966,A -85,B 0,C 180,E1 -4118.544,E2 -4118.544} C_VEL
LIN {X 0,Y 537.954,Z 443.963,A -85,B 0,C 180,E1 -4120.936,E2 -4120.936} C_VEL
LIN {X 0,Y 537.958,Z 443.965,A -85,B 0,C 180,E1 -4123.296,E2 -4123.296} C_VEL
LIN {X 0,Y 538.027,Z 443.963,A -85,B 0,C 180,E1 -4125.629,E2 -4125.629} C_VEL
LIN {X 0,Y 538.019,Z 443.959,A -85,B 0,C 180,E1 -4128.699,E2 -4128.699} C_VEL
LIN {X 0,Y 538.029,Z 443.957,A -85,B 0,C 180,E1 -4131.738,E2 -4131.738} C_VEL
LIN {X 0,Y 538.114,Z 443.951,A -85,B 0,C 180,E1 -4134.753,E2 -4134.753} C_VEL
LIN {X 0,Y 538.156,Z 443.948,A -85,B 0,C 180,E1 -4137.754,E2 -4137.754} C_VEL
LIN {X 0,Y 538.153,Z 443.946,A -85,B 0,C 180,E1 -4139.999,E2 -4139.999} C_VEL
LIN {X 0,Y 538.102,Z 443.949,A -85,B 0,C 180,E1 -4142.993,E2 -4142.993} C_VEL
LIN {X 0,Y 538.076,Z 443.963,A -85,B 0,C 180,E1 -4145.997,E2 -4145.997} C_VEL
LIN {X 0,Y 538.016,Z 443.956,A -85,B 0,C 180,E1 -4149.017,E2 -4149.017} C_VEL
LIN {X 0,Y 538.029,Z 443.965,A -85,B 0,C 180,E1 -4152.062,E2 -4152.062} C_VEL
LIN {X 0,Y 538.027,Z 443.961,A -85,B 0,C 180,E1 -4155.143,E2 -4155.143} C_VEL
LIN {X 0,Y 537.978,Z 443.966,A -85,B 0,C 180,E1 -4158.271,E2 -4158.271} C_VEL
LIN {X 0,Y 537.991,Z 443.964,A -85,B 0,C 180,E1 -4160.652,E2 -4160.652} C_VEL
LIN {X 0,Y 537.995,Z 443.965,A -85,B 0,C 180,E1 -4163.071,E2 -4163.071} C_VEL
LIN {X 0,Y 537.976,Z 443.97,A -85,B 0,C 180,E1 -4165.659,E2 -4165.659} C_VEL
LIN {X 0,Y 537.961,Z 443.972,A -85,B 0,C 180,E1 -4168.053,E2 -4168.053} C_VEL
LIN {X 0,Y 537.989,Z 443.967,A -85,B 0,C 180,E1 -4170.627,E2 -4170.627} C_VEL
LIN {X 0,Y 538.007,Z 443.962,A -85,B 0,C 180,E1 -4173.277,E2 -4173.277} C_VEL
LIN {X 0,Y 537.942,Z 443.977,A -85,B 0,C 180,E1 -4176.007,E2 -4176.007} C_VEL
LIN {X 0,Y 537.993,Z 443.965,A -85,B 0,C 180,E1 -4178.83,E2 -4178.83} C_VEL
LIN {X 0,Y 537.971,Z 443.967,A -85,B 0,C 180,E1 -4180.228,E2 -4180.228} C_VEL
LIN {X 0,Y 537.306,Z 444.049,A -85,B 0,C 180,E1 -4180.853,E2 -4180.853} C_VEL
LIN {X 0,Y 534.45,Z 444.41,A -85,B 0,C 180,E1 -4181.868,E2 -4181.868} C_VEL
LIN {X 0,Y 532.034,Z 444.713,A -85,B 0,C 180,E1 -4182.685,E2 -4182.685} C_VEL
LIN {X 0,Y 530.994,Z 444.84,A -85,B 0,C 180,E1 -4183.316,E2 -4183.316} C_VEL
LIN {X 0,Y 530.909,Z 444.849,A -85,B 0,C 180,E1 -4183.529,E2 -4183.529} C_VEL
LIN {X 0,Y 530.949,Z 444.844,A -85,B 0,C 180,E1 -4185.623,E2 -4185.623} C_VEL
LIN {X 0,Y 530.893,Z 444.844,A -85,B 0,C 180,E1 -4188.555,E2 -4188.555} C_VEL
LIN {X 0,Y 530.93,Z 444.847,A -85,B 0,C 180,E1 -4191.528,E2 -4191.528} C_VEL
LIN {X 0,Y 530.912,Z 444.844,A -85,B 0,C 180,E1 -4194.377,E2 -4194.377} C_VEL
LIN {X 0,Y 530.937,Z 444.843,A -85,B 0,C 180,E1 -4197.132,E2 -4197.132} C_VEL
LIN {X 0,Y 530.93,Z 444.851,A -85,B 0,C 180,E1 -4199.801,E2 -4199.801} C_VEL
LIN {X 0,Y 530.938,Z 444.848,A -85,B 0,C 180,E1 -4202.479,E2 -4202.479} C_VEL
LIN {X 0,Y 530.928,Z 444.846,A -85,B 0,C 180,E1 -4204.939,E2 -4204.939} C_VEL
LIN {X 0,Y 530.959,Z 444.85,A -85,B 0,C 180,E1 -4207.898,E2 -4207.898} C_VEL
LIN {X 0,Y 530.951,Z 444.845,A -85,B 0,C 180,E1 -4210.676,E2 -4210.676} C_VEL
LIN {X 0,Y 530.918,Z 444.848,A -85,B 0,C 180,E1 -4213.069,E2 -4213.069} C_VEL
LIN {X 0,Y 530.989,Z 444.841,A -85,B 0,C 180,E1 -4215.435,E2 -4215.435} C_VEL
LIN {X 0,Y 530.969,Z 444.844,A -85,B 0,C 180,E1 -4218.548,E2 -4218.548} C_VEL
LIN {X 0,Y 530.971,Z 444.845,A -85,B 0,C 180,E1 -4221.628,E2 -4221.628} C_VEL
LIN {X 0,Y 531.067,Z 444.831,A -85,B 0,C 180,E1 -4224.685,E2 -4224.685} C_VEL
LIN {X 0,Y 531.118,Z 444.829,A -85,B 0,C 180,E1 -4227.725,E2 -4227.725} C_VEL
LIN {X 0,Y 531.112,Z 444.832,A -85,B 0,C 180,E1 -4230,E2 -4230} C_VEL
LIN {X 0,Y 531.118,Z 444.829,A -85,B 0,C 180,E1 -4232.275,E2 -4232.275} C_VEL
LIN {X 0,Y 531.067,Z 444.831,A -85,B 0,C 180,E1 -4235.315,E2 -4235.315} C_VEL
LIN {X 0,Y 530.971,Z 444.845,A -85,B 0,C 180,E1 -4238.372,E2 -4238.372} C_VEL
LIN {X 0,Y 530.994,Z 444.843,A -85,B 0,C 180,E1 -4241.651,E2 -4241.651} C_VEL
LIN {X 0,Y 531.006,Z 444.837,A -85,B 0,C 180,E1 -4244.952,E2 -4244.952} C_VEL
LIN {X 0,Y 530.954,Z 444.849,A -85,B 0,C 180,E1 -4247.724,E2 -4247.724} C_VEL
LIN {X 0,Y 530.996,Z 444.845,A -85,B 0,C 180,E1 -4250.128,E2 -4250.128} C_VEL
LIN {X 0,Y 530.923,Z 444.849,A -85,B 0,C 180,E1 -4252.574,E2 -4252.574} C_VEL
LIN {X 0,Y 530.928,Z 444.846,A -85,B 0,C 180,E1 -4255.061,E2 -4255.061} C_VEL
LIN {X 0,Y 530.934,Z 444.849,A -85,B 0,C 180,E1 -4257.6,E2 -4257.6} C_VEL
LIN {X 0,Y 530.939,Z 444.845,A -85,B 0,C 180,E1 -4260.642,E2 -4260.642} C_VEL
LIN {X 0,Y 530.933,Z 444.848,A -85,B 0,C 180,E1 -4263.776,E2 -4263.776} C_VEL
LIN {X 0,Y 530.89,Z 444.851,A -85,B 0,C 180,E1 -4266.563,E2 -4266.563} C_VEL
LIN {X 0,Y 530.934,Z 444.846,A -85,B 0,C 180,E1 -4269.448,E2 -4269.448} C_VEL
LIN {X 0,Y 530.896,Z 444.843,A -85,B 0,C 180,E1 -4272.464,E2 -4272.464} C_VEL
LIN {X 0,Y 530.948,Z 444.843,A -85,B 0,C 180,E1 -4275.451,E2 -4275.451} C_VEL
LIN {X 0,Y 530.94,Z 444.842,A -85,B 0,C 180,E1 -4278.562,E2 -4278.562} C_VEL
LIN {X 0,Y 530.935,Z 444.847,A -85,B 0,C 180,E1 -4281.53,E2 -4281.53} C_VEL
LIN {X 0,Y 530.914,Z 444.846,A -85,B 0,C 180,E1 -4284.379,E2 -4284.379} C_VEL
LIN {X 0,Y 530.941,Z 444.842,A -85,B 0,C 180,E1 -4287.133,E2 -4287.133} C_VEL
LIN {X 0,Y 530.934,Z 444.852,A -85,B 0,C 180,E1 -4289.803,E2 -4289.803} C_VEL
LIN {X 0,Y 530.943,Z 444.839,A -85,B 0,C 180,E1 -4292.481,E2 -4292.481} C_VEL
LIN {X 0,Y 530.933,Z 444.843,A -85,B 0,C 180,E1 -4294.94,E2 -4294.94} C_VEL
LIN {X 0,Y 530.966,Z 444.848,A -85,B 0,C 180,E1 -4297.9,E2 -4297.9} C_VEL
LIN {X 0,Y 530.928,Z 444.838,A -85,B 0,C 180,E1 -4300.676,E2 -4300.676} C_VEL
LIN {X 0,Y 530.919,Z 444.844,A -85,B 0,C 180,E1 -4303.07,E2 -4303.07} C_VEL
LIN {X 0,Y 530.991,Z 444.84,A -85,B 0,C 180,E1 -4305.436,E2 -4305.436} C_VEL
LIN {X 0,Y 530.977,Z 444.834,A -85,B 0,C 180,E1 -4308.55,E2 -4308.55} C_VEL
LIN {X 0,Y 530.974,Z 444.838,A -85,B 0,C 180,E1 -4311.629,E2 -4311.629} C_VEL
LIN {X 0,Y 531.075,Z 444.827,A -85,B 0,C 180,E1 -4314.686,E2 -4314.686} C_VEL
LIN {X 0,Y 531.126,Z 444.824,A -85,B 0,C 180,E1 -4317.726,E2 -4317.726} C_VEL
LIN {X 0,Y 531.121,Z 444.821,A -85,B 0,C 180,E1 -4320.001,E2 -4320.001} C_VEL
LIN {X 0,Y 531.127,Z 444.823,A -85,B 0,C 180,E1 -4322.276,E2 -4322.276} C_VEL
LIN {X 0,Y 531.075,Z 444.828,A -85,B 0,C 180,E1 -4325.316,E2 -4325.316} C_VEL
LIN {X 0,Y 530.977,Z 444.833,A -85,B 0,C 180,E1 -4328.373,E2 -4328.373} C_VEL
LIN {X 0,Y 531.007,Z 444.836,A -85,B 0,C 180,E1 -4331.651,E2 -4331.651} C_VEL
LIN {X 0,Y 530.959,Z 444.84,A -85,B 0,C 180,E1 -4334.929,E2 -4334.929} C_VEL
LIN {X 0,Y 530.966,Z 444.842,A -85,B 0,C 180,E1 -4337.725,E2 -4337.725} C_VEL
LIN {X 0,Y 530.931,Z 444.843,A -85,B 0,C 180,E1 -4340.942,E2 -4340.942} C_VEL
LIN {X 0,Y 530.946,Z 444.845,A -85,B 0,C 180,E1 -4343.398,E2 -4343.398} C_VEL
LIN {X 0,Y 530.941,Z 444.845,A -85,B 0,C 180,E1 -4345.902,E2 -4345.902} C_VEL
LIN {X 0,Y 530.927,Z 444.846,A -85,B 0,C 180,E1 -4348.461,E2 -4348.461} C_VEL
LIN {X 0,Y 530.941,Z 444.844,A -85,B 0,C 180,E1 -4351.081,E2 -4351.081} C_VEL
LIN {X 0,Y 530.947,Z 444.846,A -85,B 0,C 180,E1 -4353.776,E2 -4353.776} C_VEL
LIN {X 0,Y 530.904,Z 444.849,A -85,B 0,C 180,E1 -4356.563,E2 -4356.563} C_VEL
LIN {X 0,Y 530.938,Z 444.845,A -85,B 0,C 180,E1 -4359.449,E2 -4359.449} C_VEL
LIN {X 0,Y 530.903,Z 444.85,A -85,B 0,C 180,E1 -4362.465,E2 -4362.465} C_VEL
LIN {X 0,Y 530.961,Z 444.844,A -85,B 0,C 180,E1 -4365.451,E2 -4365.451} C_VEL
LIN {X 0,Y 530.908,Z 444.842,A -85,B 0,C 180,E1 -4368.557,E2 -4368.557} C_VEL
LIN {X 0,Y 530.945,Z 444.847,A -85,B 0,C 180,E1 -4371.529,E2 -4371.529} C_VEL
LIN {X 0,Y 530.926,Z 444.848,A -85,B 0,C 180,E1 -4374.378,E2 -4374.378} C_VEL
LIN {X 0,Y 530.946,Z 444.842,A -85,B 0,C 180,E1 -4377.132,E2 -4377.132} C_VEL
LIN {X 0,Y 530.944,Z 444.85,A -85,B 0,C 180,E1 -4379.802,E2 -4379.802} C_VEL
LIN {X 0,Y 530.954,Z 444.848,A -85,B 0,C 180,E1 -4382.481,E2 -4382.481} C_VEL
LIN {X 0,Y 531.007,Z 445.056,A -85,B 0,C 180,E1 -4384.159,E2 -4384.159} C_VEL
LIN {X 0,Y 532.127,Z 452.309,A -85,B 0,C 180,E1 -4385.688,E2 -4385.688} C_VEL
LIN {X 0,Y 531.751,Z 467.553,A -85,B 0,C 180,E1 -4388.687,E2 -4388.687} C_VEL
LIN {X 0,Y 531.47,Z 483.35,A -85,B 0,C 180,E1 -4391.716,E2 -4391.716} C_VEL
LIN {X 0,Y 531.126,Z 500.961,A -85,B 0,C 180,E1 -4395.023,E2 -4395.023} C_VEL
LIN {X 0,Y 531.588,Z 503.987,A -85,B 0,C 180,E1 -4395.117,E2 -4395.117} C_VEL
LIN {X 0,Y 532.79,Z 511.103,A -85,B 0,C 180,E1 -4395.248,E2 -4395.248} C_VEL
LIN {X 0,Y 532.39,Z 605.941,A -85,B 0,C 180,E1 -4396.546,E2 -4396.546} C_VEL
LIN {X 0,Y 532.331,Z 615.863,A -85,B 0,C 180,E1 -4396.763,E2 -4396.763} C_VEL
LIN {X 0,Y 532.169,Z 625.854,A -85,B 0,C 180,E1 -4397.075,E2 -4397.075} C_VEL
LIN {X 0,Y 531.957,Z 636.215,A -85,B 0,C 180,E1 -4397.506,E2 -4397.506} C_VEL
LIN {X 0,Y 531.785,Z 645.68,A -85,B 0,C 180,E1 -4398.005,E2 -4398.005} C_VEL
LIN {X 0,Y 531.629,Z 654.375,A -85,B 0,C 180,E1 -4398.563,E2 -4398.563} C_VEL
LIN {X 0,Y 531.372,Z 663.105,A -85,B 0,C 180,E1 -4399.233,E2 -4399.233} C_VEL
LIN {X 0,Y 531.199,Z 670.53,A -85,B 0,C 180,E1 -4399.904,E2 -4399.904} C_VEL
LIN {X 0,Y 530.937,Z 679.328,A -85,B 0,C 180,E1 -4400.86,E2 -4400.86} C_VEL
LIN {X 0,Y 530.846,Z 685.297,A -85,B 0,C 180,E1 -4401.626,E2 -4401.626} C_VEL
LIN {X 0,Y 530.684,Z 691.579,A -85,B 0,C 180,E1 -4402.581,E2 -4402.581} C_VEL
LIN {X 0,Y 530.548,Z 697.58,A -85,B 0,C 180,E1 -4403.697,E2 -4403.697} C_VEL
LIN {X 0,Y 530.523,Z 701.886,A -85,B 0,C 180,E1 -4404.679,E2 -4404.679} C_VEL
LIN {X 0,Y 530.523,Z 705.822,A -85,B 0,C 180,E1 -4405.822,E2 -4405.822} C_VEL
LIN {X 0,Y 530.457,Z 708.734,A -85,B 0,C 180,E1 -4406.962,E2 -4406.962} C_VEL
LIN {X 0,Y 530.411,Z 710.215,A -85,B 0,C 180,E1 -4407.722,E2 -4407.722} C_VEL
LIN {X 0,Y 530.344,Z 711.729,A -85,B 0,C 180,E1 -4409.241,E2 -4409.241} C_VEL
LIN {X 0,Y 530.343,Z 712,A -85,B 0,C 180,E1 -4410,E2 -4410} C_VEL
LIN {X 0,Y 530.361,Z 711.14,A -85,B 0,C 180,E1 -4411.519,E2 -4411.519} C_VEL
LIN {X 0,Y 530.411,Z 710.215,A -85,B 0,C 180,E1 -4412.278,E2 -4412.278} C_VEL
LIN {X 0,Y 530.516,Z 706.903,A -85,B 0,C 180,E1 -4413.798,E2 -4413.798} C_VEL
LIN {X 0,Y 530.458,Z 703.304,A -85,B 0,C 180,E1 -4414.94,E2 -4414.94} C_VEL
LIN {X 0,Y 530.606,Z 700.382,A -85,B 0,C 180,E1 -4415.701,E2 -4415.701} C_VEL
LIN {X 0,Y 530.638,Z 694.839,A -85,B 0,C 180,E1 -4416.846,E2 -4416.846} C_VEL
LIN {X 0,Y 530.759,Z 689.215,A -85,B 0,C 180,E1 -4417.8,E2 -4417.8} C_VEL
LIN {X 0,Y 530.926,Z 682.441,A -85,B 0,C 180,E1 -4418.756,E2 -4418.756} C_VEL
LIN {X 0,Y 531.094,Z 674.232,A -85,B 0,C 180,E1 -4419.713,E2 -4419.713} C_VEL
LIN {X 0,Y 531.28,Z 666.402,A -85,B 0,C 180,E1 -4420.48,E2 -4420.48} C_VEL
LIN {X 0,Y 531.518,Z 658.315,A -85,B 0,C 180,E1 -4421.15,E2 -4421.15} C_VEL
LIN {X 0,Y 531.741,Z 648.123,A -85,B 0,C 180,E1 -4421.847,E2 -4421.847} C_VEL
LIN {X 0,Y 531.889,Z 640.154,A -85,B 0,C 180,E1 -4422.302,E2 -4422.302} C_VEL
LIN {X 0,Y 532.073,Z 629.642,A -85,B 0,C 180,E1 -4422.782,E2 -4422.782} C_VEL
LIN {X 0,Y 532.268,Z 619.307,A -85,B 0,C 180,E1 -4423.141,E2 -4423.141} C_VEL
LIN {X 0,Y 532.389,Z 608.585,A -85,B 0,C 180,E1 -4423.405,E2 -4423.405} C_VEL
LIN {X 0,Y 532.567,Z 585.812,A -85,B 0,C 180,E1 -4423.741,E2 -4423.741} C_VEL
LIN {X 0,Y 532.743,Z 510.419,A -85,B 0,C 180,E1 -4424.763,E2 -4424.763} C_VEL
LIN {X 0,Y 531.136,Z 501.301,A -85,B 0,C 180,E1 -4424.952,E2 -4424.952} C_VEL
LIN {X 0,Y 531.151,Z 500.025,A -85,B 0,C 180,E1 -4425.126,E2 -4425.126} C_VEL
LIN {X 0,Y 531.455,Z 482.199,A -85,B 0,C 180,E1 -4428.504,E2 -4428.504} C_VEL
LIN {X 0,Y 531.751,Z 467.553,A -85,B 0,C 180,E1 -4431.313,E2 -4431.313} C_VEL
LIN {X 0,Y 532.108,Z 453.061,A -85,B 0,C 180,E1 -4434.17,E2 -4434.17} C_VEL
LIN {X 0,Y 531.721,Z 448.89,A -85,B 0,C 180,E1 -4435.021,E2 -4435.021} C_VEL
LIN {X 0,Y 530.974,Z 444.931,A -85,B 0,C 180,E1 -4435.899,E2 -4435.899} C_VEL
LIN {X 0,Y 530.93,Z 444.851,A -85,B 0,C 180,E1 -4438.459,E2 -4438.459} C_VEL
LIN {X 0,Y 530.94,Z 444.846,A -85,B 0,C 180,E1 -4441.08,E2 -4441.08} C_VEL
LIN {X 0,Y 530.951,Z 444.846,A -85,B 0,C 180,E1 -4443.775,E2 -4443.775} C_VEL
LIN {X 0,Y 530.904,Z 444.851,A -85,B 0,C 180,E1 -4446.562,E2 -4446.562} C_VEL
LIN {X 0,Y 530.949,Z 444.844,A -85,B 0,C 180,E1 -4449.446,E2 -4449.446} C_VEL
LIN {X 0,Y 530.911,Z 444.851,A -85,B 0,C 180,E1 -4452.463,E2 -4452.463} C_VEL
LIN {X 0,Y 530.96,Z 444.842,A -85,B 0,C 180,E1 -4455.449,E2 -4455.449} C_VEL
LIN {X 0,Y 530.907,Z 444.85,A -85,B 0,C 180,E1 -4458.555,E2 -4458.555} C_VEL
LIN {X 0,Y 530.929,Z 444.845,A -85,B 0,C 180,E1 -4461.526,E2 -4461.526} C_VEL
LIN {X 0,Y 530.926,Z 444.848,A -85,B 0,C 180,E1 -4464.377,E2 -4464.377} C_VEL
LIN {X 0,Y 530.952,Z 444.839,A -85,B 0,C 180,E1 -4467.131,E2 -4467.131} C_VEL
LIN {X 0,Y 530.944,Z 444.848,A -85,B 0,C 180,E1 -4469.801,E2 -4469.801} C_VEL
LIN {X 0,Y 530.951,Z 444.839,A -85,B 0,C 180,E1 -4472.479,E2 -4472.479} C_VEL
LIN {X 0,Y 530.941,Z 444.841,A -85,B 0,C 180,E1 -4474.938,E2 -4474.938} C_VEL
LIN {X 0,Y 530.974,Z 444.845,A -85,B 0,C 180,E1 -4477.898,E2 -4477.898} C_VEL
LIN {X 0,Y 530.912,Z 444.841,A -85,B 0,C 180,E1 -4480.673,E2 -4480.673} C_VEL
LIN {X 0,Y 530.923,Z 444.841,A -85,B 0,C 180,E1 -4483.068,E2 -4483.068} C_VEL
LIN {X 0,Y 530.976,Z 444.839,A -85,B 0,C 180,E1 -4485.434,E2 -4485.434} C_VEL
LIN {X 0,Y 530.981,Z 444.836,A -85,B 0,C 180,E1 -4488.547,E2 -4488.547} C_VEL
LIN {X 0,Y 530.977,Z 444.833,A -85,B 0,C 180,E1 -4491.627,E2 -4491.627} C_VEL
LIN {X 0,Y 531.075,Z 444.828,A -85,B 0,C 180,E1 -4494.684,E2 -4494.684} C_VEL
LIN {X 0,Y 531.127,Z 444.823,A -85,B 0,C 180,E1 -4497.724,E2 -4497.724} C_VEL
LIN {X 0,Y 531.121,Z 444.821,A -85,B 0,C 180,E1 -4499.999,E2 -4499.999} C_VEL
LIN {X 0,Y 531.126,Z 444.824,A -85,B 0,C 180,E1 -4502.274,E2 -4502.274} C_VEL
LIN {X 0,Y 531.075,Z 444.827,A -85,B 0,C 180,E1 -4505.314,E2 -4505.314} C_VEL
LIN {X 0,Y 530.974,Z 444.838,A -85,B 0,C 180,E1 -4508.371,E2 -4508.371} C_VEL
LIN {X 0,Y 531.002,Z 444.833,A -85,B 0,C 180,E1 -4511.649,E2 -4511.649} C_VEL
LIN {X 0,Y 531.01,Z 444.835,A -85,B 0,C 180,E1 -4514.949,E2 -4514.949} C_VEL
LIN {X 0,Y 530.96,Z 444.843,A -85,B 0,C 180,E1 -4517.723,E2 -4517.723} C_VEL
LIN {X 0,Y 530.963,Z 444.838,A -85,B 0,C 180,E1 -4520.938,E2 -4520.938} C_VEL
LIN {X 0,Y 530.942,Z 444.853,A -85,B 0,C 180,E1 -4524.03,E2 -4524.03} C_VEL
LIN {X 0,Y 530.932,Z 444.84,A -85,B 0,C 180,E1 -4526.746,E2 -4526.746} C_VEL
LIN {X 0,Y 530.948,Z 444.841,A -85,B 0,C 180,E1 -4529.323,E2 -4529.323} C_VEL
LIN {X 0,Y 530.94,Z 444.851,A -85,B 0,C 180,E1 -4532.097,E2 -4532.097} C_VEL
LIN {X 0,Y 530.942,Z 444.839,A -85,B 0,C 180,E1 -4534.848,E2 -4534.848} C_VEL
LIN {X 0,Y 530.915,Z 444.849,A -85,B 0,C 180,E1 -4537.51,E2 -4537.51} C_VEL
LIN {X 0,Y 530.933,Z 444.845,A -85,B 0,C 180,E1 -4540.435,E2 -4540.435} C_VEL
LIN {X 0,Y 530.909,Z 444.849,A -85,B 0,C 180,E1 -4543.529,E2 -4543.529} C_VEL
LIN {X 0,Y 530.245,Z 444.936,A -85,B 0,C 180,E1 -4544.163,E2 -4544.163} C_VEL
LIN {X 0,Y 527.407,Z 445.282,A -85,B 0,C 180,E1 -4545.192,E2 -4545.192} C_VEL
LIN {X 0,Y 524.999,Z 445.585,A -85,B 0,C 180,E1 -4546.021,E2 -4546.021} C_VEL
LIN {X 0,Y 523.953,Z 445.707,A -85,B 0,C 180,E1 -4546.66,E2 -4546.66} C_VEL
LIN {X 0,Y 523.861,Z 445.716,A -85,B 0,C 180,E1 -4546.877,E2 -4546.877} C_VEL
LIN {X 0,Y 523.857,Z 445.726,A -85,B 0,C 180,E1 -4549.913,E2 -4549.913} C_VEL
LIN {X 0,Y 523.852,Z 445.727,A -85,B 0,C 180,E1 -4552.864,E2 -4552.864} C_VEL
LIN {X 0,Y 523.894,Z 445.718,A -85,B 0,C 180,E1 -4555.707,E2 -4555.707} C_VEL
LIN {X 0,Y 523.892,Z 445.725,A -85,B 0,C 180,E1 -4558.454,E2 -4558.454} C_VEL
LIN {X 0,Y 523.881,Z 445.719,A -85,B 0,C 180,E1 -4561.122,E2 -4561.122} C_VEL
LIN {X 0,Y 523.891,Z 445.731,A -85,B 0,C 180,E1 -4563.997,E2 -4563.997} C_VEL
LIN {X 0,Y 523.89,Z 445.729,A -85,B 0,C 180,E1 -4566.269,E2 -4566.269} C_VEL
LIN {X 0,Y 523.921,Z 445.72,A -85,B 0,C 180,E1 -4568.766,E2 -4568.766} C_VEL
LIN {X 0,Y 523.911,Z 445.721,A -85,B 0,C 180,E1 -4571.219,E2 -4571.219} C_VEL
LIN {X 0,Y 523.895,Z 445.726,A -85,B 0,C 180,E1 -4574.437,E2 -4574.437} C_VEL
LIN {X 0,Y 523.929,Z 445.722,A -85,B 0,C 180,E1 -4577.607,E2 -4577.607} C_VEL
LIN {X 0,Y 523.958,Z 445.716,A -85,B 0,C 180,E1 -4580.738,E2 -4580.738} C_VEL
LIN {X 0,Y 523.989,Z 445.718,A -85,B 0,C 180,E1 -4583.84,E2 -4583.84} C_VEL
LIN {X 0,Y 524.088,Z 445.704,A -85,B 0,C 180,E1 -4587.694,E2 -4587.694} C_VEL
LIN {X 0,Y 524.08,Z 445.707,A -85,B 0,C 180,E1 -4590,E2 -4590} C_VEL
LIN {X 0,Y 524.088,Z 445.704,A -85,B 0,C 180,E1 -4592.306,E2 -4592.306} C_VEL
LIN {X 0,Y 523.989,Z 445.718,A -85,B 0,C 180,E1 -4596.16,E2 -4596.16} C_VEL
LIN {X 0,Y 523.958,Z 445.716,A -85,B 0,C 180,E1 -4599.262,E2 -4599.262} C_VEL
LIN {X 0,Y 523.929,Z 445.722,A -85,B 0,C 180,E1 -4602.393,E2 -4602.393} C_VEL
LIN {X 0,Y 523.895,Z 445.727,A -85,B 0,C 180,E1 -4605.563,E2 -4605.563} C_VEL
LIN {X 0,Y 523.911,Z 445.721,A -85,B 0,C 180,E1 -4608.781,E2 -4608.781} C_VEL
LIN {X 0,Y 523.921,Z 445.72,A -85,B 0,C 180,E1 -4611.234,E2 -4611.234} C_VEL
LIN {X 0,Y 523.915,Z 445.726,A -85,B 0,C 180,E1 -4614.196,E2 -4614.196} C_VEL
LIN {X 0,Y 523.876,Z 445.725,A -85,B 0,C 180,E1 -4617.137,E2 -4617.137} C_VEL
LIN {X 0,Y 523.877,Z 445.724,A -85,B 0,C 180,E1 -4619.76,E2 -4619.76} C_VEL
LIN {X 0,Y 523.883,Z 445.725,A -85,B 0,C 180,E1 -4622.453,E2 -4622.453} C_VEL
LIN {X 0,Y 523.89,Z 445.715,A -85,B 0,C 180,E1 -4625.229,E2 -4625.229} C_VEL
LIN {X 0,Y 523.883,Z 445.73,A -85,B 0,C 180,E1 -4628.104,E2 -4628.104} C_VEL
LIN {X 0,Y 523.861,Z 445.719,A -85,B 0,C 180,E1 -4631.301,E2 -4631.301} C_VEL
LIN {X 0,Y 523.918,Z 445.717,A -85,B 0,C 180,E1 -4634.69,E2 -4634.69} C_VEL
LIN {X 0,Y 523.881,Z 445.731,A -85,B 0,C 180,E1 -4637.876,E2 -4637.876} C_VEL
LIN {X 0,Y 523.896,Z 445.721,A -85,B 0,C 180,E1 -4640.915,E2 -4640.915} C_VEL
LIN {X 0,Y 523.843,Z 445.735,A -85,B 0,C 180,E1 -4643.823,E2 -4643.823} C_VEL
LIN {X 0,Y 523.896,Z 445.721,A -85,B 0,C 180,E1 -4646.634,E2 -4646.634} C_VEL
LIN {X 0,Y 523.926,Z 445.719,A -85,B 0,C 180,E1 -4649.356,E2 -4649.356} C_VEL
LIN {X 0,Y 523.9,Z 445.718,A -85,B 0,C 180,E1 -4652.297,E2 -4652.297} C_VEL
LIN {X 0,Y 523.889,Z 445.723,A -85,B 0,C 180,E1 -4655.428,E2 -4655.428} C_VEL
LIN {X 0,Y 523.926,Z 445.724,A -85,B 0,C 180,E1 -4657.941,E2 -4657.941} C_VEL
LIN {X 0,Y 523.915,Z 445.713,A -85,B 0,C 180,E1 -4660.407,E2 -4660.407} C_VEL
LIN {X 0,Y 523.885,Z 445.72,A -85,B 0,C 180,E1 -4662.836,E2 -4662.836} C_VEL
LIN {X 0,Y 523.953,Z 445.715,A -85,B 0,C 180,E1 -4665.236,E2 -4665.236} C_VEL
LIN {X 0,Y 523.951,Z 445.71,A -85,B 0,C 180,E1 -4668.394,E2 -4668.394} C_VEL
LIN {X 0,Y 523.937,Z 445.713,A -85,B 0,C 180,E1 -4671.516,E2 -4671.516} C_VEL
LIN {X 0,Y 524.022,Z 445.706,A -85,B 0,C 180,E1 -4674.614,E2 -4674.614} C_VEL
LIN {X 0,Y 524.096,Z 445.699,A -85,B 0,C 180,E1 -4677.696,E2 -4677.696} C_VEL
LIN {X 0,Y 524.09,Z 445.695,A -85,B 0,C 180,E1 -4680.001,E2 -4680.001} C_VEL
LIN {X 0,Y 524.097,Z 445.699,A -85,B 0,C 180,E1 -4682.307,E2 -4682.307} C_VEL
LIN {X 0,Y 523.995,Z 445.712,A -85,B 0,C 180,E1 -4686.161,E2 -4686.161} C_VEL
LIN {X 0,Y 523.938,Z 445.707,A -85,B 0,C 180,E1 -4689.264,E2 -4689.264} C_VEL
LIN {X 0,Y 523.941,Z 445.717,A -85,B 0,C 180,E1 -4692.394,E2 -4692.394} C_VEL
LIN {X 0,Y 523.878,Z 445.726,A -85,B 0,C 180,E1 -4695.565,E2 -4695.565} C_VEL
LIN {X 0,Y 523.9,Z 445.719,A -85,B 0,C 180,E1 -4697.972,E2 -4697.972} C_VEL
LIN {X 0,Y 523.902,Z 445.721,A -85,B 0,C 180,E1 -4700.414,E2 -4700.414} C_VEL
LIN {X 0,Y 523.904,Z 445.72,A -85,B 0,C 180,E1 -4702.895,E2 -4702.895} C_VEL
LIN {X 0,Y 523.892,Z 445.721,A -85,B 0,C 180,E1 -4705.423,E2 -4705.423} C_VEL
LIN {X 0,Y 523.893,Z 445.726,A -85,B 0,C 180,E1 -4708.004,E2 -4708.004} C_VEL
LIN {X 0,Y 523.906,Z 445.72,A -85,B 0,C 180,E1 -4710.849,E2 -4710.849} C_VEL
LIN {X 0,Y 523.924,Z 445.72,A -85,B 0,C 180,E1 -4713.73,E2 -4713.73} C_VEL
LIN {X 0,Y 523.858,Z 445.729,A -85,B 0,C 180,E1 -4716.395,E2 -4716.395} C_VEL
LIN {X 0,Y 523.892,Z 445.72,A -85,B 0,C 180,E1 -4719.088,E2 -4719.088} C_VEL
LIN {X 0,Y 523.885,Z 445.728,A -85,B 0,C 180,E1 -4722.126,E2 -4722.126} C_VEL
LIN {X 0,Y 523.932,Z 445.718,A -85,B 0,C 180,E1 -4725.312,E2 -4725.312} C_VEL
LIN {X 0,Y 523.876,Z 445.717,A -85,B 0,C 180,E1 -4728.701,E2 -4728.701} C_VEL
LIN {X 0,Y 523.898,Z 445.73,A -85,B 0,C 180,E1 -4731.897,E2 -4731.897} C_VEL
LIN {X 0,Y 523.889,Z 445.722,A -85,B 0,C 180,E1 -4734.918,E2 -4734.918} C_VEL
LIN {X 0,Y 523.9,Z 445.725,A -85,B 0,C 180,E1 -4737.687,E2 -4737.687} C_VEL
LIN {X 0,Y 523.905,Z 445.724,A -85,B 0,C 180,E1 -4740.687,E2 -4740.687} C_VEL
LIN {X 0,Y 523.902,Z 445.728,A -85,B 0,C 180,E1 -4743.725,E2 -4743.725} C_VEL
LIN {X 0,Y 523.955,Z 445.932,A -85,B 0,C 180,E1 -4743.988,E2 -4743.988} C_VEL
LIN {X 0,Y 525.182,Z 453.589,A -85,B 0,C 180,E1 -4745.625,E2 -4745.625} C_VEL
LIN {X 0,Y 524.784,Z 469.51,A -85,B 0,C 180,E1 -4748.802,E2 -4748.802} C_VEL
LIN {X 0,Y 524.387,Z 486.243,A -85,B 0,C 180,E1 -4752.046,E2 -4752.046} C_VEL
LIN {X 0,Y 524.132,Z 500.923,A -85,B 0,C 180,E1 -4754.832,E2 -4754.832} C_VEL
LIN {X 0,Y 525.64,Z 510,A -85,B 0,C 180,E1 -4755.03,E2 -4755.03} C_VEL
LIN {X 0,Y 525.914,Z 514.657,A -85,B 0,C 180,E1 -4755.102,E2 -4755.102} C_VEL
LIN {X 0,Y 525.504,Z 605.745,A -85,B 0,C 180,E1 -4756.366,E2 -4756.366} C_VEL
LIN {X 0,Y 525.409,Z 615.666,A -85,B 0,C 180,E1 -4756.586,E2 -4756.586} C_VEL
LIN {X 0,Y 525.246,Z 625.658,A -85,B 0,C 180,E1 -4756.901,E2 -4756.901} C_VEL
LIN {X 0,Y 525.003,Z 636.018,A -85,B 0,C 180,E1 -4757.338,E2 -4757.338} C_VEL
LIN {X 0,Y 524.831,Z 645.351,A -85,B 0,C 180,E1 -4757.836,E2 -4757.836} C_VEL
LIN {X 0,Y 524.64,Z 654.178,A -85,B 0,C 180,E1 -4758.408,E2 -4758.408} C_VEL
LIN {X 0,Y 524.359,Z 662.908,A -85,B 0,C 180,E1 -4759.087,E2 -4759.087} C_VEL
LIN {X 0,Y 524.171,Z 670.333,A -85,B 0,C 180,E1 -4759.767,E2 -4759.767} C_VEL
LIN {X 0,Y 523.911,Z 679.131,A -85,B 0,C 180,E1 -4760.737,E2 -4760.737} C_VEL
LIN {X 0,Y 523.786,Z 685.124,A -85,B 0,C 180,E1 -4761.513,E2 -4761.513} C_VEL
LIN {X 0,Y 523.633,Z 691.434,A -85,B 0,C 180,E1 -4762.481,E2 -4762.481} C_VEL
LIN {X 0,Y 523.524,Z 696.579,A -85,B 0,C 180,E1 -4763.42,E2 -4763.42} C_VEL
LIN {X 0,Y 523.462,Z 701.797,A -85,B 0,C 180,E1 -4764.607,E2 -4764.607} C_VEL
LIN {X 0,Y 523.425,Z 705.756,A -85,B 0,C 180,E1 -4765.765,E2 -4765.765} C_VEL
LIN {X 0,Y 523.368,Z 708.683,A -85,B 0,C 180,E1 -4766.921,E2 -4766.921} C_VEL
LIN {X 0,Y 523.335,Z 710.179,A -85,B 0,C 180,E1 -4767.691,E2 -4767.691} C_VEL
LIN {X 0,Y 523.25,Z 711.695,A -85,B 0,C 180,E1 -4769.23,E2 -4769.23} C_VEL
LIN {X 0,Y 523.246,Z 711.973,A -85,B 0,C 180,E1 -4770,E2 -4770} C_VEL
LIN {X 0,Y 523.275,Z 711.102,A -85,B 0,C 180,E1 -4771.539,E2 -4771.539} C_VEL
LIN {X 0,Y 523.335,Z 710.179,A -85,B 0,C 180,E1 -4772.309,E2 -4772.309} C_VEL
LIN {X 0,Y 523.444,Z 706.844,A -85,B 0,C 180,E1 -4773.849,E2 -4773.849} C_VEL
LIN {X 0,Y 523.383,Z 703.221,A -85,B 0,C 180,E1 -4775.007,E2 -4775.007} C_VEL
LIN {X 0,Y 523.517,Z 700.285,A -85,B 0,C 180,E1 -4775.779,E2 -4775.779} C_VEL
LIN {X 0,Y 523.576,Z 694.711,A -85,B 0,C 180,E1 -4776.939,E2 -4776.939} C_VEL
LIN {X 0,Y 523.688,Z 689.059,A -85,B 0,C 180,E1 -4777.906,E2 -4777.906} C_VEL
LIN {X 0,Y 523.843,Z 682.254,A -85,B 0,C 180,E1 -4778.875,E2 -4778.875} C_VEL
LIN {X 0,Y 524.049,Z 674.034,A -85,B 0,C 180,E1 -4779.845,E2 -4779.845} C_VEL
LIN {X 0,Y 524.293,Z 666.205,A -85,B 0,C 180,E1 -4780.621,E2 -4780.621} C_VEL
LIN {X 0,Y 524.523,Z 658.118,A -85,B 0,C 180,E1 -4781.301,E2 -4781.301} C_VEL
LIN {X 0,Y 524.749,Z 648.944,A -85,B 0,C 180,E1 -4781.945,E2 -4781.945} C_VEL
LIN {X 0,Y 524.946,Z 639.957,A -85,B 0,C 180,E1 -4782.467,E2 -4782.467} C_VEL
LIN {X 0,Y 525.156,Z 629.446,A -85,B 0,C 180,E1 -4782.953,E2 -4782.953} C_VEL
LIN {X 0,Y 525.355,Z 619.111,A -85,B 0,C 180,E1 -4783.317,E2 -4783.317} C_VEL
LIN {X 0,Y 525.468,Z 608.389,A -85,B 0,C 180,E1 -4783.585,E2 -4783.585} C_VEL
LIN {X 0,Y 525.677,Z 585.615,A -85,B 0,C 180,E1 -4783.925,E2 -4783.925} C_VEL
LIN {X 0,Y 525.805,Z 510.914,A -85,B 0,C 180,E1 -4784.953,E2 -4784.953} C_VEL
LIN {X 0,Y 524.123,Z 501.005,A -85,B 0,C 180,E1 -4785.162,E2 -4785.162} C_VEL
LIN {X 0,Y 524.098,Z 498.732,A -85,B 0,C 180,E1 -4785.557,E2 -4785.557} C_VEL
LIN {X 0,Y 524.474,Z 482.063,A -85,B 0,C 180,E1 -4788.76,E2 -4788.76} C_VEL
LIN {X 0,Y 524.78,Z 467.415,A -85,B 0,C 180,E1 -4791.61,E2 -4791.61} C_VEL
LIN {X 0,Y 525.168,Z 453.579,A -85,B 0,C 180,E1 -4794.378,E2 -4794.378} C_VEL
LIN {X 0,Y 523.932,Z 445.827,A -85,B 0,C 180,E1 -4796.056,E2 -4796.056} C_VEL
LIN {X 0,Y 523.874,Z 445.728,A -85,B 0,C 180,E1 -4798.878,E2 -4798.878} C_VEL
LIN {X 0,Y 523.908,Z 445.724,A -85,B 0,C 180,E1 -4801.545,E2 -4801.545} C_VEL
LIN {X 0,Y 523.912,Z 445.726,A -85,B 0,C 180,E1 -4804.291,E2 -4804.291} C_VEL
LIN {X 0,Y 523.876,Z 445.726,A -85,B 0,C 180,E1 -4807.672,E2 -4807.672} C_VEL
LIN {X 0,Y 523.883,Z 445.724,A -85,B 0,C 180,E1 -4810.122,E2 -4810.122} C_VEL
LIN {X 0,Y 523.879,Z 445.723,A -85,B 0,C 180,E1 -4813.171,E2 -4813.171} C_VEL
LIN {X 0,Y 523.915,Z 445.722,A -85,B 0,C 180,E1 -4815.769,E2 -4815.769} C_VEL
LIN {X 0,Y 523.852,Z 445.726,A -85,B 0,C 180,E1 -4818.898,E2 -4818.898} C_VEL
LIN {X 0,Y 523.888,Z 445.727,A -85,B 0,C 180,E1 -4821.895,E2 -4821.895} C_VEL
LIN {X 0,Y 523.911,Z 445.716,A -85,B 0,C 180,E1 -4824.912,E2 -4824.912} C_VEL
LIN {X 0,Y 523.9,Z 445.721,A -85,B 0,C 180,E1 -4827.685,E2 -4827.685} C_VEL
LIN {X 0,Y 523.933,Z 445.717,A -85,B 0,C 180,E1 -4830.68,E2 -4830.68} C_VEL
LIN {X 0,Y 523.887,Z 445.719,A -85,B 0,C 180,E1 -4833.723,E2 -4833.723} C_VEL
LIN {X 0,Y 523.905,Z 445.726,A -85,B 0,C 180,E1 -4836.268,E2 -4836.268} C_VEL
LIN {X 0,Y 523.903,Z 445.719,A -85,B 0,C 180,E1 -4838.764,E2 -4838.764} C_VEL
LIN {X 0,Y 523.892,Z 445.713,A -85,B 0,C 180,E1 -4841.218,E2 -4841.218} C_VEL
LIN {X 0,Y 523.868,Z 445.722,A -85,B 0,C 180,E1 -4843.636,E2 -4843.636} C_VEL
LIN {X 0,Y 523.902,Z 445.728,A -85,B 0,C 180,E1 -4846.026,E2 -4846.026} C_VEL
LIN {X 0,Y 523.955,Z 445.713,A -85,B 0,C 180,E1 -4848.392,E2 -4848.392} C_VEL
LIN {X 0,Y 523.94,Z 445.708,A -85,B 0,C 180,E1 -4851.514,E2 -4851.514} C_VEL
LIN {X 0,Y 524.022,Z 445.707,A -85,B 0,C 180,E1 -4854.612,E2 -4854.612} C_VEL
LIN {X 0,Y 524.097,Z 445.699,A -85,B 0,C 180,E1 -4857.693,E2 -4857.693} C_VEL
LIN {X 0,Y 524.09,Z 445.695,A -85,B 0,C 180,E1 -4859.999,E2 -4859.999} C_VEL
LIN {X 0,Y 524.096,Z 445.699,A -85,B 0,C 180,E1 -4862.304,E2 -4862.304} C_VEL
LIN {X 0,Y 523.998,Z 445.715,A -85,B 0,C 180,E1 -4866.158,E2 -4866.158} C_VEL
LIN {X 0,Y 523.934,Z 445.71,A -85,B 0,C 180,E1 -4869.262,E2 -4869.262} C_VEL
LIN {X 0,Y 523.937,Z 445.719,A -85,B 0,C 180,E1 -4872.392,E2 -4872.392} C_VEL
LIN {X 0,Y 523.975,Z 445.711,A -85,B 0,C 180,E1 -4875.047,E2 -4875.047} C_VEL
LIN {X 0,Y 523.897,Z 445.724,A -85,B 0,C 180,E1 -4877.97,E2 -4877.97} C_VEL
LIN {X 0,Y 523.916,Z 445.719,A -85,B 0,C 180,E1 -4880.411,E2 -4880.411} C_VEL
LIN {X 0,Y 523.896,Z 445.721,A -85,B 0,C 180,E1 -4882.893,E2 -4882.893} C_VEL
LIN {X 0,Y 523.883,Z 445.723,A -85,B 0,C 180,E1 -4885.421,E2 -4885.421} C_VEL
LIN {X 0,Y 523.884,Z 445.723,A -85,B 0,C 180,E1 -4888.002,E2 -4888.002} C_VEL
LIN {X 0,Y 523.896,Z 445.722,A -85,B 0,C 180,E1 -4890.847,E2 -4890.847} C_VEL
LIN {X 0,Y 523.913,Z 445.722,A -85,B 0,C 180,E1 -4893.728,E2 -4893.728} C_VEL
LIN {X 0,Y 523.846,Z 445.732,A -85,B 0,C 180,E1 -4896.394,E2 -4896.394} C_VEL
LIN {X 0,Y 523.896,Z 445.721,A -85,B 0,C 180,E1 -4899.085,E2 -4899.085} C_VEL
LIN {X 0,Y 523.881,Z 445.731,A -85,B 0,C 180,E1 -4902.124,E2 -4902.124} C_VEL
LIN {X 0,Y 523.918,Z 445.717,A -85,B 0,C 180,E1 -4905.31,E2 -4905.31} C_VEL
LIN {X 0,Y 523.861,Z 445.716,A -85,B 0,C 180,E1 -4906.877,E2 -4906.877} C_VEL
LIN {X 0,Y 523.17,Z 445.805,A -85,B 0,C 180,E1 -4907.518,E2 -4907.518} C_VEL
LIN {X 0,Y 520.296,Z 446.163,A -85,B 0,C 180,E1 -4908.56,E2 -4908.56} C_VEL
LIN {X 0,Y 517.894,Z 446.464,A -85,B 0,C 180,E1 -4909.398,E2 -4909.398} C_VEL
LIN {X 0,Y 516.886,Z 446.596,A -85,B 0,C 180,E1 -4910.046,E2 -4910.046} C_VEL
LIN {X 0,Y 516.815,Z 446.608,A -85,B 0,C 180,E1 -4910.265,E2 -4910.265} C_VEL
LIN {X 0,Y 516.818,Z 446.608,A -85,B 0,C 180,E1 -4912.271,E2 -4912.271} C_VEL
LIN {X 0,Y 516.854,Z 446.59,A -85,B 0,C 180,E1 -4915.173,E2 -4915.173} C_VEL
LIN {X 0,Y 516.833,Z 446.609,A -85,B 0,C 180,E1 -4917.973,E2 -4917.973} C_VEL
LIN {X 0,Y 516.886,Z 446.591,A -85,B 0,C 180,E1 -4920.694,E2 -4920.694} C_VEL
LIN {X 0,Y 516.861,Z 446.605,A -85,B 0,C 180,E1 -4923.818,E2 -4923.818} C_VEL
LIN {X 0,Y 516.839,Z 446.602,A -85,B 0,C 180,E1 -4926.775,E2 -4926.775} C_VEL
LIN {X 0,Y 516.911,Z 446.598,A -85,B 0,C 180,E1 -4929.735,E2 -4929.735} C_VEL
LIN {X 0,Y 516.851,Z 446.603,A -85,B 0,C 180,E1 -4932.594,E2 -4932.594} C_VEL
LIN {X 0,Y 516.918,Z 446.593,A -85,B 0,C 180,E1 -4935.03,E2 -4935.03} C_VEL
LIN {X 0,Y 516.908,Z 446.599,A -85,B 0,C 180,E1 -4938.232,E2 -4938.232} C_VEL
LIN {X 0,Y 516.911,Z 446.595,A -85,B 0,C 180,E1 -4941.399,E2 -4941.399} C_VEL
LIN {X 0,Y 516.965,Z 446.589,A -85,B 0,C 180,E1 -4944.539,E2 -4944.539} C_VEL
LIN {X 0,Y 517.057,Z 446.58,A -85,B 0,C 180,E1 -4947.663,E2 -4947.663} C_VEL
LIN {X 0,Y 517.049,Z 446.583,A -85,B 0,C 180,E1 -4950,E2 -4950} C_VEL
LIN {X 0,Y 517.057,Z 446.58,A -85,B 0,C 180,E1 -4952.337,E2 -4952.337} C_VEL
LIN {X 0,Y 516.955,Z 446.593,A -85,B 0,C 180,E1 -4956.244,E2 -4956.244} C_VEL
LIN {X 0,Y 516.913,Z 446.595,A -85,B 0,C 180,E1 -4959.39,E2 -4959.39} C_VEL
LIN {X 0,Y 516.882,Z 446.599,A -85,B 0,C 180,E1 -4962.565,E2 -4962.565} C_VEL
LIN {X 0,Y 516.922,Z 446.592,A -85,B 0,C 180,E1 -4965.144,E2 -4965.144} C_VEL
LIN {X 0,Y 516.858,Z 446.605,A -85,B 0,C 180,E1 -4968.224,E2 -4968.224} C_VEL
LIN {X 0,Y 516.881,Z 446.597,A -85,B 0,C 180,E1 -4970.703,E2 -4970.703} C_VEL
LIN {X 0,Y 516.839,Z 446.602,A -85,B 0,C 180,E1 -4973.225,E2 -4973.225} C_VEL
LIN {X 0,Y 516.861,Z 446.605,A -85,B 0,C 180,E1 -4976.182,E2 -4976.182} C_VEL
LIN {X 0,Y 516.868,Z 446.595,A -85,B 0,C 180,E1 -4979.519,E2 -4979.519} C_VEL
LIN {X 0,Y 516.851,Z 446.6,A -85,B 0,C 180,E1 -4982.539,E2 -4982.539} C_VEL
LIN {X 0,Y 516.833,Z 446.594,A -85,B 0,C 180,E1 -4985.328,E2 -4985.328} C_VEL
LIN {X 0,Y 516.852,Z 446.599,A -85,B 0,C 180,E1 -4988.718,E2 -4988.718} C_VEL
LIN {X 0,Y 516.817,Z 446.596,A -85,B 0,C 180,E1 -4991.784,E2 -4991.784} C_VEL
LIN {X 0,Y 516.881,Z 446.593,A -85,B 0,C 180,E1 -4995.008,E2 -4995.008} C_VEL
LIN {X 0,Y 516.838,Z 446.599,A -85,B 0,C 180,E1 -4998.408,E2 -4998.408} C_VEL
LIN {X 0,Y 516.859,Z 446.598,A -85,B 0,C 180,E1 -5001.284,E2 -5001.284} C_VEL
LIN {X 0,Y 516.836,Z 446.596,A -85,B 0,C 180,E1 -5004.674,E2 -5004.674} C_VEL
LIN {X 0,Y 516.855,Z 446.599,A -85,B 0,C 180,E1 -5007.463,E2 -5007.463} C_VEL
LIN {X 0,Y 516.873,Z 446.596,A -85,B 0,C 180,E1 -5010.483,E2 -5010.483} C_VEL
LIN {X 0,Y 516.821,Z 446.597,A -85,B 0,C 180,E1 -5013.338,E2 -5013.338} C_VEL
LIN {X 0,Y 516.873,Z 446.604,A -85,B 0,C 180,E1 -5015.928,E2 -5015.928} C_VEL
LIN {X 0,Y 516.864,Z 446.596,A -85,B 0,C 180,E1 -5018.463,E2 -5018.463} C_VEL
LIN {X 0,Y 516.85,Z 446.589,A -85,B 0,C 180,E1 -5020.954,E2 -5020.954} C_VEL
LIN {X 0,Y 516.821,Z 446.602,A -85,B 0,C 180,E1 -5023.409,E2 -5023.409} C_VEL
LIN {X 0,Y 516.863,Z 446.605,A -85,B 0,C 180,E1 -5025.834,E2 -5025.834} C_VEL
LIN {X 0,Y 516.917,Z 446.588,A -85,B 0,C 180,E1 -5028.234,E2 -5028.234} C_VEL
LIN {X 0,Y 516.911,Z 446.586,A -85,B 0,C 180,E1 -5031.4,E2 -5031.4} C_VEL
LIN {X 0,Y 516.973,Z 446.585,A -85,B 0,C 180,E1 -5034.541,E2 -5034.541} C_VEL
LIN {X 0,Y 517.066,Z 446.575,A -85,B 0,C 180,E1 -5037.664,E2 -5037.664} C_VEL
LIN {X 0,Y 517.059,Z 446.57,A -85,B 0,C 180,E1 -5040.001,E2 -5040.001} C_VEL
LIN {X 0,Y 517.067,Z 446.574,A -85,B 0,C 180,E1 -5042.338,E2 -5042.338} C_VEL
LIN {X 0,Y 516.962,Z 446.586,A -85,B 0,C 180,E1 -5046.245,E2 -5046.245} C_VEL
LIN {X 0,Y 516.9,Z 446.584,A -85,B 0,C 180,E1 -5049.391,E2 -5049.391} C_VEL
LIN {X 0,Y 516.894,Z 446.593,A -85,B 0,C 180,E1 -5052.566,E2 -5052.566} C_VEL
LIN {X 0,Y 516.824,Z 446.608,A -85,B 0,C 180,E1 -5055.782,E2 -5055.782} C_VEL
LIN {X 0,Y 516.843,Z 446.596,A -85,B 0,C 180,E1 -5058.226,E2 -5058.226} C_VEL
LIN {X 0,Y 516.863,Z 446.595,A -85,B 0,C 180,E1 -5060.705,E2 -5060.705} C_VEL
LIN {X 0,Y 516.853,Z 446.599,A -85,B 0,C 180,E1 -5063.225,E2 -5063.225} C_VEL
LIN {X 0,Y 516.866,Z 446.594,A -85,B 0,C 180,E1 -5066.18,E2 -5066.18} C_VEL
LIN {X 0,Y 516.901,Z 446.593,A -85,B 0,C 180,E1 -5069.307,E2 -5069.307} C_VEL
LIN {X 0,Y 516.847,Z 446.603,A -85,B 0,C 180,E1 -5072.028,E2 -5072.028} C_VEL
LIN {X 0,Y 516.868,Z 446.593,A -85,B 0,C 180,E1 -5074.827,E2 -5074.827} C_VEL
LIN {X 0,Y 516.85,Z 446.606,A -85,B 0,C 180,E1 -5077.94,E2 -5077.94} C_VEL
LIN {X 0,Y 516.819,Z 446.602,A -85,B 0,C 180,E1 -5080.749,E2 -5080.749} C_VEL
LIN {X 0,Y 516.86,Z 446.604,A -85,B 0,C 180,E1 -5083.907,E2 -5083.907} C_VEL
LIN {X 0,Y 516.86,Z 446.604,A -85,B 0,C 180,E1 -5086.111,E2 -5086.111} C_VEL
LIN {X 0,Y 516.82,Z 446.597,A -85,B 0,C 180,E1 -5089.253,E2 -5089.253} C_VEL
LIN {X 0,Y 516.858,Z 446.604,A -85,B 0,C 180,E1 -5092.061,E2 -5092.061} C_VEL
LIN {X 0,Y 516.853,Z 446.6,A -85,B 0,C 180,E1 -5095.173,E2 -5095.173} C_VEL
LIN {X 0,Y 516.848,Z 446.607,A -85,B 0,C 180,E1 -5097.974,E2 -5097.974} C_VEL
LIN {X 0,Y 516.874,Z 446.6,A -85,B 0,C 180,E1 -5100.693,E2 -5100.693} C_VEL
LIN {X 0,Y 516.883,Z 446.74,A -85,B 0,C 180,E1 -5103.791,E2 -5103.791} C_VEL
LIN {X 0,Y 518.126,Z 453.791,A -85,B 0,C 180,E1 -5105.342,E2 -5105.342} C_VEL
LIN {X 0,Y 517.951,Z 463.492,A -85,B 0,C 180,E1 -5107.323,E2 -5107.323} C_VEL
LIN {X 0,Y 517.622,Z 476.117,A -85,B 0,C 180,E1 -5109.836,E2 -5109.836} C_VEL
LIN {X 0,Y 517.282,Z 490.283,A -85,B 0,C 180,E1 -5112.609,E2 -5112.609} C_VEL
LIN {X 0,Y 517.046,Z 500.596,A -85,B 0,C 180,E1 -5114.609,E2 -5114.609} C_VEL
LIN {X 0,Y 517.923,Z 505.865,A -85,B 0,C 180,E1 -5114.747,E2 -5114.747} C_VEL
LIN {X 0,Y 519.061,Z 513.681,A -85,B 0,C 180,E1 -5114.89,E2 -5114.89} C_VEL
LIN {X 0,Y 518.627,Z 605.549,A -85,B 0,C 180,E1 -5116.182,E2 -5116.182} C_VEL
LIN {X 0,Y 518.507,Z 615.47,A -85,B 0,C 180,E1 -5116.404,E2 -5116.404} C_VEL
LIN {X 0,Y 518.312,Z 625.461,A -85,B 0,C 180,E1 -5116.723,E2 -5116.723} C_VEL
LIN {X 0,Y 518.052,Z 635.821,A -85,B 0,C 180,E1 -5117.165,E2 -5117.165} C_VEL
LIN {X 0,Y 517.872,Z 645.024,A -85,B 0,C 180,E1 -5117.662,E2 -5117.662} C_VEL
LIN {X 0,Y 517.65,Z 653.981,A -85,B 0,C 180,E1 -5118.25,E2 -5118.25} C_VEL
LIN {X 0,Y 517.361,Z 662.711,A -85,B 0,C 180,E1 -5118.938,E2 -5118.938} C_VEL
LIN {X 0,Y 517.15,Z 670.136,A -85,B 0,C 180,E1 -5119.627,E2 -5119.627} C_VEL
LIN {X 0,Y 516.868,Z 678.934,A -85,B 0,C 180,E1 -5120.609,E2 -5120.609} C_VEL
LIN {X 0,Y 516.738,Z 684.927,A -85,B 0,C 180,E1 -5121.396,E2 -5121.396} C_VEL
LIN {X 0,Y 516.563,Z 691.237,A -85,B 0,C 180,E1 -5122.377,E2 -5122.377} C_VEL
LIN {X 0,Y 516.422,Z 696.916,A -85,B 0,C 180,E1 -5123.447,E2 -5123.447} C_VEL
LIN {X 0,Y 516.378,Z 701.6,A -85,B 0,C 180,E1 -5124.533,E2 -5124.533} C_VEL
LIN {X 0,Y 516.313,Z 705.559,A -85,B 0,C 180,E1 -5125.707,E2 -5125.707} C_VEL
LIN {X 0,Y 516.283,Z 708.487,A -85,B 0,C 180,E1 -5126.879,E2 -5126.879} C_VEL
LIN {X 0,Y 516.262,Z 709.983,A -85,B 0,C 180,E1 -5127.659,E2 -5127.659} C_VEL
LIN {X 0,Y 516.16,Z 711.499,A -85,B 0,C 180,E1 -5129.22,E2 -5129.22} C_VEL
LIN {X 0,Y 516.154,Z 711.777,A -85,B 0,C 180,E1 -5130,E2 -5130} C_VEL
LIN {X 0,Y 516.192,Z 710.906,A -85,B 0,C 180,E1 -5131.56,E2 -5131.56} C_VEL
LIN {X 0,Y 516.262,Z 709.983,A -85,B 0,C 180,E1 -5132.341,E2 -5132.341} C_VEL
LIN {X 0,Y 516.353,Z 706.647,A -85,B 0,C 180,E1 -5133.902,E2 -5133.902} C_VEL
LIN {X 0,Y 516.313,Z 703.025,A -85,B 0,C 180,E1 -5135.076,E2 -5135.076} C_VEL
LIN {X 0,Y 516.427,Z 700.088,A -85,B 0,C 180,E1 -5135.858,E2 -5135.858} C_VEL
LIN {X 0,Y 516.508,Z 694.514,A -85,B 0,C 180,E1 -5137.034,E2 -5137.034} C_VEL
LIN {X 0,Y 516.641,Z 688.862,A -85,B 0,C 180,E1 -5138.015,E2 -5138.015} C_VEL
LIN {X 0,Y 516.792,Z 682.057,A -85,B 0,C 180,E1 -5138.997,E2 -5138.997} C_VEL
LIN {X 0,Y 517.024,Z 673.837,A -85,B 0,C 180,E1 -5139.98,E2 -5139.98} C_VEL
LIN {X 0,Y 517.284,Z 666.008,A -85,B 0,C 180,E1 -5140.767,E2 -5140.767} C_VEL
LIN {X 0,Y 517.557,Z 657.922,A -85,B 0,C 180,E1 -5141.455,E2 -5141.455} C_VEL
LIN {X 0,Y 517.765,Z 648.039,A -85,B 0,C 180,E1 -5142.152,E2 -5142.152} C_VEL
LIN {X 0,Y 518.009,Z 639.761,A -85,B 0,C 180,E1 -5142.637,E2 -5142.637} C_VEL
LIN {X 0,Y 518.242,Z 629.25,A -85,B 0,C 180,E1 -5143.129,E2 -5143.129} C_VEL
LIN {X 0,Y 518.45,Z 618.915,A -85,B 0,C 180,E1 -5143.498,E2 -5143.498} C_VEL
LIN {X 0,Y 518.577,Z 608.193,A -85,B 0,C 180,E1 -5143.769,E2 -5143.769} C_VEL
LIN {X 0,Y 518.78,Z 585.419,A -85,B 0,C 180,E1 -5144.114,E2 -5144.114} C_VEL
LIN {X 0,Y 518.944,Z 511.779,A -85,B 0,C 180,E1 -5145.14,E2 -5145.14} C_VEL
LIN {X 0,Y 517.108,Z 501.03,A -85,B 0,C 180,E1 -5145.359,E2 -5145.359} C_VEL
LIN {X 0,Y 517.05,Z 499.651,A -85,B 0,C 180,E1 -5145.549,E2 -5145.549} C_VEL
LIN {X 0,Y 517.443,Z 484.017,A -85,B 0,C 180,E1 -5148.613,E2 -5148.613} C_VEL
LIN {X 0,Y 517.814,Z 468.324,A -85,B 0,C 180,E1 -5151.706,E2 -5151.706} C_VEL
LIN {X 0,Y 518.207,Z 455.36,A -85,B 0,C 180,E1 -5154.331,E2 -5154.331} C_VEL
LIN {X 0,Y 517.456,Z 449.675,A -85,B 0,C 180,E1 -5155.545,E2 -5155.545} C_VEL
LIN {X 0,Y 516.901,Z 446.708,A -85,B 0,C 180,E1 -5156.239,E2 -5156.239} C_VEL
LIN {X 0,Y 516.862,Z 446.602,A -85,B 0,C 180,E1 -5159.513,E2 -5159.513} C_VEL
LIN {X 0,Y 516.892,Z 446.596,A -85,B 0,C 180,E1 -5162.541,E2 -5162.541} C_VEL
LIN {X 0,Y 516.849,Z 446.6,A -85,B 0,C 180,E1 -5165.326,E2 -5165.326} C_VEL
LIN {X 0,Y 516.868,Z 446.598,A -85,B 0,C 180,E1 -5168.717,E2 -5168.717} C_VEL
LIN {X 0,Y 516.832,Z 446.598,A -85,B 0,C 180,E1 -5171.783,E2 -5171.783} C_VEL
LIN {X 0,Y 516.897,Z 446.592,A -85,B 0,C 180,E1 -5175.006,E2 -5175.006} C_VEL
LIN {X 0,Y 516.828,Z 446.605,A -85,B 0,C 180,E1 -5178.409,E2 -5178.409} C_VEL
LIN {X 0,Y 516.858,Z 446.596,A -85,B 0,C 180,E1 -5181.281,E2 -5181.281} C_VEL
LIN {X 0,Y 516.848,Z 446.598,A -85,B 0,C 180,E1 -5184.672,E2 -5184.672} C_VEL
LIN {X 0,Y 516.866,Z 446.595,A -85,B 0,C 180,E1 -5187.461,E2 -5187.461} C_VEL
LIN {X 0,Y 516.883,Z 446.597,A -85,B 0,C 180,E1 -5190.481,E2 -5190.481} C_VEL
LIN {X 0,Y 516.829,Z 446.594,A -85,B 0,C 180,E1 -5193.336,E2 -5193.336} C_VEL
LIN {X 0,Y 516.881,Z 446.599,A -85,B 0,C 180,E1 -5195.926,E2 -5195.926} C_VEL
LIN {X 0,Y 516.857,Z 446.599,A -85,B 0,C 180,E1 -5198.46,E2 -5198.46} C_VEL
LIN {X 0,Y 516.842,Z 446.591,A -85,B 0,C 180,E1 -5200.952,E2 -5200.952} C_VEL
LIN {X 0,Y 516.825,Z 446.597,A -85,B 0,C 180,E1 -5203.406,E2 -5203.406} C_VEL
LIN {X 0,Y 516.853,Z 446.603,A -85,B 0,C 180,E1 -5205.831,E2 -5205.831} C_VEL
LIN {X 0,Y 516.922,Z 446.591,A -85,B 0,C 180,E1 -5208.232,E2 -5208.232} C_VEL
LIN {X 0,Y 516.914,Z 446.582,A -85,B 0,C 180,E1 -5211.398,E2 -5211.398} C_VEL
LIN {X 0,Y 516.973,Z 446.586,A -85,B 0,C 180,E1 -5214.538,E2 -5214.538} C_VEL
LIN {X 0,Y 517.067,Z 446.574,A -85,B 0,C 180,E1 -5217.662,E2 -5217.662} C_VEL
LIN {X 0,Y 517.059,Z 446.57,A -85,B 0,C 180,E1 -5219.999,E2 -5219.999} C_VEL
LIN {X 0,Y 517.066,Z 446.575,A -85,B 0,C 180,E1 -5222.336,E2 -5222.336} C_VEL
LIN {X 0,Y 516.964,Z 446.59,A -85,B 0,C 180,E1 -5226.242,E2 -5226.242} C_VEL
LIN {X 0,Y 516.897,Z 446.587,A -85,B 0,C 180,E1 -5229.389,E2 -5229.389} C_VEL
LIN {X 0,Y 516.89,Z 446.595,A -85,B 0,C 180,E1 -5232.564,E2 -5232.564} C_VEL
LIN {X 0,Y 516.927,Z 446.589,A -85,B 0,C 180,E1 -5235.141,E2 -5235.141} C_VEL
LIN {X 0,Y 516.841,Z 446.597,A -85,B 0,C 180,E1 -5238.224,E2 -5238.224} C_VEL
LIN {X 0,Y 516.874,Z 446.594,A -85,B 0,C 180,E1 -5240.702,E2 -5240.702} C_VEL
LIN {X 0,Y 516.845,Z 446.6,A -85,B 0,C 180,E1 -5243.223,E2 -5243.223} C_VEL
LIN {X 0,Y 516.856,Z 446.599,A -85,B 0,C 180,E1 -5246.178,E2 -5246.178} C_VEL
LIN {X 0,Y 516.89,Z 446.592,A -85,B 0,C 180,E1 -5249.305,E2 -5249.305} C_VEL
LIN {X 0,Y 516.837,Z 446.609,A -85,B 0,C 180,E1 -5252.026,E2 -5252.026} C_VEL
LIN {X 0,Y 516.857,Z 446.594,A -85,B 0,C 180,E1 -5254.825,E2 -5254.825} C_VEL
LIN {X 0,Y 516.845,Z 446.608,A -85,B 0,C 180,E1 -5257.939,E2 -5257.939} C_VEL
LIN {X 0,Y 516.836,Z 446.597,A -85,B 0,C 180,E1 -5260.744,E2 -5260.744} C_VEL
LIN {X 0,Y 516.866,Z 446.605,A -85,B 0,C 180,E1 -5263.903,E2 -5263.903} C_VEL
LIN {X 0,Y 516.813,Z 446.593,A -85,B 0,C 180,E1 -5266.879,E2 -5266.879} C_VEL
LIN {X 0,Y 516.816,Z 446.598,A -85,B 0,C 180,E1 -5269.596,E2 -5269.596} C_VEL
LIN {X 0,Y 516.815,Z 446.608,A -85,B 0,C 180,E1 -5270.265,E2 -5270.265} C_VEL
LIN {X 0,Y 516.176,Z 446.7,A -85,B 0,C 180,E1 -5270.915,E2 -5270.915} C_VEL
LIN {X 0,Y 513.318,Z 447.061,A -85,B 0,C 180,E1 -5271.971,E2 -5271.971} C_VEL
LIN {X 0,Y 510.883,Z 447.358,A -85,B 0,C 180,E1 -5272.821,E2 -5272.821} C_VEL
LIN {X 0,Y 509.834,Z 447.479,A -85,B 0,C 180,E1 -5273.478,E2 -5273.478} C_VEL
LIN {X 0,Y 509.749,Z 447.486,A -85,B 0,C 180,E1 -5273.7,E2 -5273.7} C_VEL
LIN {X 0,Y 509.817,Z 447.476,A -85,B 0,C 180,E1 -5276.536,E2 -5276.536} C_VEL
LIN {X 0,Y 509.811,Z 447.477,A -85,B 0,C 180,E1 -5279.332,E2 -5279.332} C_VEL
LIN {X 0,Y 509.808,Z 447.482,A -85,B 0,C 180,E1 -5282.05,E2 -5282.05} C_VEL
LIN {X 0,Y 509.782,Z 447.482,A -85,B 0,C 180,E1 -5284.699,E2 -5284.699} C_VEL
LIN {X 0,Y 509.808,Z 447.48,A -85,B 0,C 180,E1 -5287.458,E2 -5287.458} C_VEL
LIN {X 0,Y 509.889,Z 447.474,A -85,B 0,C 180,E1 -5289.844,E2 -5289.844} C_VEL
LIN {X 0,Y 509.83,Z 447.48,A -85,B 0,C 180,E1 -5292.346,E2 -5292.346} C_VEL
LIN {X 0,Y 509.868,Z 447.471,A -85,B 0,C 180,E1 -5294.818,E2 -5294.818} C_VEL
LIN {X 0,Y 509.872,Z 447.477,A -85,B 0,C 180,E1 -5298.131,E2 -5298.131} C_VEL
LIN {X 0,Y 509.865,Z 447.472,A -85,B 0,C 180,E1 -5301.279,E2 -5301.279} C_VEL
LIN {X 0,Y 509.903,Z 447.471,A -85,B 0,C 180,E1 -5303.67,E2 -5303.67} C_VEL
LIN {X 0,Y 509.868,Z 447.472,A -85,B 0,C 180,E1 -5306.839,E2 -5306.839} C_VEL
LIN {X 0,Y 509.905,Z 447.47,A -85,B 0,C 180,E1 -5308.42,E2 -5308.42} C_VEL
LIN {X 0,Y 510.017,Z 447.459,A -85,B 0,C 180,E1 -5310,E2 -5310} C_VEL
LIN {X 0,Y 510.025,Z 447.455,A -85,B 0,C 180,E1 -5312.369,E2 -5312.369} C_VEL
LIN {X 0,Y 509.92,Z 447.468,A -85,B 0,C 180,E1 -5315.536,E2 -5315.536} C_VEL
LIN {X 0,Y 509.859,Z 447.479,A -85,B 0,C 180,E1 -5317.923,E2 -5317.923} C_VEL
LIN {X 0,Y 509.845,Z 447.474,A -85,B 0,C 180,E1 -5321.127,E2 -5321.127} C_VEL
LIN {X 0,Y 509.828,Z 447.479,A -85,B 0,C 180,E1 -5323.553,E2 -5323.553} C_VEL
LIN {X 0,Y 509.785,Z 447.488,A -85,B 0,C 180,E1 -5326.005,E2 -5326.005} C_VEL
LIN {X 0,Y 509.817,Z 447.48,A -85,B 0,C 180,E1 -5328.485,E2 -5328.485} C_VEL
LIN {X 0,Y 509.824,Z 447.476,A -85,B 0,C 180,E1 -5331.003,E2 -5331.003} C_VEL
LIN {X 0,Y 509.8,Z 447.482,A -85,B 0,C 180,E1 -5333.565,E2 -5333.565} C_VEL
LIN {X 0,Y 509.797,Z 447.483,A -85,B 0,C 180,E1 -5336.357,E2 -5336.357} C_VEL
LIN {X 0,Y 509.816,Z 447.471,A -85,B 0,C 180,E1 -5338.848,E2 -5338.848} C_VEL
LIN {X 0,Y 509.786,Z 447.483,A -85,B 0,C 180,E1 -5341.592,E2 -5341.592} C_VEL
LIN {X 0,Y 509.816,Z 447.469,A -85,B 0,C 180,E1 -5344.416,E2 -5344.416} C_VEL
LIN {X 0,Y 509.763,Z 447.483,A -85,B 0,C 180,E1 -5347.345,E2 -5347.345} C_VEL
LIN {X 0,Y 509.77,Z 447.475,A -85,B 0,C 180,E1 -5350.388,E2 -5350.388} C_VEL
LIN {X 0,Y 509.777,Z 447.473,A -85,B 0,C 180,E1 -5353.576,E2 -5353.576} C_VEL
LIN {X 0,Y 509.79,Z 447.481,A -85,B 0,C 180,E1 -5356.427,E2 -5356.427} C_VEL
LIN {X 0,Y 509.799,Z 447.477,A -85,B 0,C 180,E1 -5359.616,E2 -5359.616} C_VEL
LIN {X 0,Y 509.766,Z 447.483,A -85,B 0,C 180,E1 -5362.657,E2 -5362.657} C_VEL
LIN {X 0,Y 509.825,Z 447.474,A -85,B 0,C 180,E1 -5365.802,E2 -5365.802} C_VEL
LIN {X 0,Y 509.824,Z 447.475,A -85,B 0,C 180,E1 -5368.723,E2 -5368.723} C_VEL
LIN {X 0,Y 509.821,Z 447.472,A -85,B 0,C 180,E1 -5371.154,E2 -5371.154} C_VEL
LIN {X 0,Y 509.825,Z 447.474,A -85,B 0,C 180,E1 -5373.826,E2 -5373.826} C_VEL
LIN {X 0,Y 509.807,Z 447.479,A -85,B 0,C 180,E1 -5376.437,E2 -5376.437} C_VEL
LIN {X 0,Y 509.83,Z 447.474,A -85,B 0,C 180,E1 -5379.614,E2 -5379.614} C_VEL
LIN {X 0,Y 509.835,Z 447.473,A -85,B 0,C 180,E1 -5382.348,E2 -5382.348} C_VEL
LIN {X 0,Y 509.876,Z 447.468,A -85,B 0,C 180,E1 -5384.819,E2 -5384.819} C_VEL
LIN {X 0,Y 509.881,Z 447.465,A -85,B 0,C 180,E1 -5388.132,E2 -5388.132} C_VEL
LIN {X 0,Y 509.864,Z 447.463,A -85,B 0,C 180,E1 -5391.28,E2 -5391.28} C_VEL
LIN {X 0,Y 509.912,Z 447.467,A -85,B 0,C 180,E1 -5393.671,E2 -5393.671} C_VEL
LIN {X 0,Y 509.876,Z 447.465,A -85,B 0,C 180,E1 -5396.841,E2 -5396.841} C_VEL
LIN {X 0,Y 509.914,Z 447.455,A -85,B 0,C 180,E1 -5398.422,E2 -5398.422} C_VEL
LIN {X 0,Y 510.027,Z 447.445,A -85,B 0,C 180,E1 -5400.001,E2 -5400.001} C_VEL
LIN {X 0,Y 510.035,Z 447.45,A -85,B 0,C 180,E1 -5402.37,E2 -5402.37} C_VEL
LIN {X 0,Y 509.929,Z 447.465,A -85,B 0,C 180,E1 -5405.537,E2 -5405.537} C_VEL
LIN {X 0,Y 509.869,Z 447.467,A -85,B 0,C 180,E1 -5407.924,E2 -5407.924} C_VEL
LIN {X 0,Y 509.857,Z 447.464,A -85,B 0,C 180,E1 -5411.128,E2 -5411.128} C_VEL
LIN {X 0,Y 509.817,Z 447.477,A -85,B 0,C 180,E1 -5413.554,E2 -5413.554} C_VEL
LIN {X 0,Y 509.785,Z 447.481,A -85,B 0,C 180,E1 -5416.006,E2 -5416.006} C_VEL
LIN {X 0,Y 509.805,Z 447.469,A -85,B 0,C 180,E1 -5418.487,E2 -5418.487} C_VEL
LIN {X 0,Y 509.814,Z 447.473,A -85,B 0,C 180,E1 -5421.004,E2 -5421.004} C_VEL
LIN {X 0,Y 509.815,Z 447.479,A -85,B 0,C 180,E1 -5423.565,E2 -5423.565} C_VEL
LIN {X 0,Y 509.804,Z 447.471,A -85,B 0,C 180,E1 -5426.355,E2 -5426.355} C_VEL
LIN {X 0,Y 509.831,Z 447.472,A -85,B 0,C 180,E1 -5428.848,E2 -5428.848} C_VEL
LIN {X 0,Y 509.801,Z 447.482,A -85,B 0,C 180,E1 -5431.592,E2 -5431.592} C_VEL
LIN {X 0,Y 509.831,Z 447.472,A -85,B 0,C 180,E1 -5434.416,E2 -5434.416} C_VEL
LIN {X 0,Y 509.775,Z 447.482,A -85,B 0,C 180,E1 -5437.345,E2 -5437.345} C_VEL
LIN {X 0,Y 509.785,Z 447.481,A -85,B 0,C 180,E1 -5440.388,E2 -5440.388} C_VEL
LIN {X 0,Y 509.791,Z 447.483,A -85,B 0,C 180,E1 -5443.576,E2 -5443.576} C_VEL
LIN {X 0,Y 509.792,Z 447.48,A -85,B 0,C 180,E1 -5446.426,E2 -5446.426} C_VEL
